# B&R Automation Studio project PLC code - cp (part 3)

#### Alarms.st
```iecst
ACTION Alarms:

	IF EDGEPOS(gDryer.AlSummary.xAlarmCritical) THEN
		MpAlarmXSet(gAlrCore, 'Dryer.Alarm.GenCritical');
	ELSIF EDGENEG(gDryer.AlSummary.xAlarmCritical) THEN
		MpAlarmXReset(gAlrCore, 'Dryer.Alarm.GenCritical');
	END_IF

	IF EDGEPOS(gDryer.AlSummary.xAlarmStop) THEN
		MpAlarmXSet(gAlrCore, 'Dryer.Alarm.GenStop');
	ELSIF EDGENEG(gDryer.AlSummary.xAlarmStop) THEN
		MpAlarmXReset(gAlrCore, 'Dryer.Alarm.GenStop');
	END_IF

	IF EDGEPOS(gDryer.Al.xAlrStopDrying) THEN
		MpAlarmXSet(gAlrCore, 'Dryer.Alarm.GenStopDrying');
	ELSIF EDGENEG(gDryer.Al.xAlrStopDrying) THEN
		MpAlarmXReset(gAlrCore, 'Dryer.Alarm.GenStopDrying');
	END_IF

	IF EDGEPOS(gDryer.Al.Alarm.xFanBreakers) THEN
		MpAlarmXSet(gAlrCore, 'Dryer.Alarm.FanBreakers');
	ELSIF EDGENEG(gDryer.Al.Alarm.xFanBreakers) THEN
		MpAlarmXReset(gAlrCore, 'Dryer.Alarm.FanBreakers');
	END_IF

	IF EDGEPOS(gDryer.Al.Alarm.xFan24Vdc) THEN
		MpAlarmXSet(gAlrCore, 'Dryer.Alarm.FansPsu');
	ELSIF EDGENEG(gDryer.Al.Alarm.xFan24Vdc) THEN
		MpAlarmXReset(gAlrCore, 'Dryer.Alarm.FansPsu');
	END_IF

	IF EDGEPOS(gDryer.Al.Alarm.xMain24Vdc) THEN
		MpAlarmXSet(gAlrCore, 'Dryer.Alarm.MainPsu');
	ELSIF EDGENEG(gDryer.Al.Alarm.xMain24Vdc) THEN
		MpAlarmXReset(gAlrCore, 'Dryer.Alarm.MainPsu');
	END_IF

	IF EDGEPOS(gDryer.Al.Alarm.xAlarmMountedMedia) THEN
		MpAlarmXSet(gAlrCore, 'Dryer.Alarm.MountedMedia');
	ELSIF EDGENEG(gDryer.Al.Alarm.xAlarmMountedMedia) THEN
		MpAlarmXReset(gAlrCore, 'Dryer.Alarm.MountedMedia');
	END_IF

	IF EDGEPOS(gDryer.Al.Alarm.Safety.xEStopFront) THEN
		MpAlarmXSet(gAlrCore, 'Dryer.Alarm.EstopFront');
	ELSIF EDGENEG(gDryer.Al.Alarm.Safety.xEStopFront) THEN
		MpAlarmXReset(gAlrCore, 'Dryer.Alarm.EstopFront');
	END_IF

	IF EDGEPOS(gDryer.Al.Alarm.Safety.xEStopRear) THEN
		MpAlarmXSet(gAlrCore, 'Dryer.Alarm.EstopRear');
	ELSIF EDGENEG(gDryer.Al.Alarm.Safety.xEStopRear) THEN
		MpAlarmXReset(gAlrCore, 'Dryer.Alarm.EstopRear');
	END_IF

	IF EDGEPOS(gDryer.Al.Alarm.Safety.xRemoteEStop) THEN
		MpAlarmXSet(gAlrCore, 'Dryer.Alarm.EstopRemote');
	ELSIF EDGENEG(gDryer.Al.Alarm.Safety.xRemoteEStop) THEN
		MpAlarmXReset(gAlrCore, 'Dryer.Alarm.EstopRemote');
	END_IF

	IF EDGEPOS(gDryer.Al.Alarm.xAlrWrongPhysConf) THEN
		MpAlarmXSet(gAlrCore, 'Dryer.Alarm.WrongPhysConfig');
	ELSIF EDGENEG(gDryer.Al.Alarm.xAlrWrongPhysConf) THEN
		MpAlarmXReset(gAlrCore, 'Dryer.Alarm.WrongPhysConfig');
	END_IF

	IF EDGEPOS(gDryer.Al.Alarm.xAlrBeltOvertorque) THEN
		MpAlarmXSet(gAlrCore, 'Dryer.Alarm.OvertorqueBelt');
	ELSIF EDGENEG(gDryer.Al.Alarm.xAlrBeltOvertorque) THEN
		MpAlarmXReset(gAlrCore, 'Dryer.Alarm.OvertorqueBelt');
	END_IF

	IF EDGEPOS(gDryer.Al.Alarm.xAlrBeltOverTempFast) THEN
		MpAlarmXSet(gAlrCore, 'Dryer.Alarm.OverTempBeltFast');
	ELSIF EDGENEG(gDryer.Al.Alarm.xAlrBeltOverTempFast) THEN
		MpAlarmXReset(gAlrCore, 'Dryer.Alarm.OverTempBeltFast');
	END_IF

	IF EDGEPOS(gDryer.Al.Alarm.xAlrBeltOverTempSlow) THEN
		MpAlarmXSet(gAlrCore, 'Dryer.Alarm.OverTempBeltSlow');
	ELSIF EDGENEG(gDryer.Al.Alarm.xAlrBeltOverTempSlow) THEN
		MpAlarmXReset(gAlrCore, 'Dryer.Alarm.OverTempBeltSlow');
	END_IF

	IF EDGEPOS(gDryer.Al.Warning.xFanBreakersHighLoad) THEN
		MpAlarmXSet(gAlrCore, 'Dryer.Alarm.FansPsu80');
	ELSIF EDGENEG(gDryer.Al.Warning.xFanBreakersHighLoad) THEN
		MpAlarmXReset(gAlrCore, 'Dryer.Alarm.FansPsu80');
	END_IF

	IF EDGEPOS(gDryer.Al.Warning.xMountedMediaInside) THEN
		MpAlarmXSet(gAlrCore, 'Dryer.Warning.MountedMediaInside');
	ELSIF EDGENEG(gDryer.Al.Warning.xMountedMediaInside) THEN
		MpAlarmXReset(gAlrCore, 'Dryer.Warning.MountedMediaInside');
	END_IF

	IF EDGEPOS(gDryer.Al.Warning.xBeltSensorError) THEN
		MpAlarmXSet(gAlrCore, 'Dryer.Warning.BeltTempSensError');
	ELSIF EDGENEG(gDryer.Al.Warning.xBeltSensorError) THEN
		MpAlarmXReset(gAlrCore, 'Dryer.Warning.BeltTempSensError');
	END_IF

	IF EDGEPOS(gDryer.Al.Warning.xBoardInSensorError) THEN
		MpAlarmXSet(gAlrCore, 'Dryer.Warning.BoardInTempSensError');
	ELSIF EDGENEG(gDryer.Al.Warning.xBoardInSensorError) THEN
		MpAlarmXReset(gAlrCore, 'Dryer.Warning.BoardInTempSensError');
	END_IF

	IF EDGEPOS(gDryer.Al.Warning.xBoardOutSensorError) THEN
		MpAlarmXSet(gAlrCore, 'Dryer.Warning.BoardOutTempSensError');
	ELSIF EDGENEG(gDryer.Al.Warning.xBoardOutSensorError) THEN
		MpAlarmXReset(gAlrCore, 'Dryer.Warning.BoardOutTempSensError');
	END_IF

	IF EDGEPOS(gDryer.Al.Warning.xAirBlowerInputSensorError) THEN
		MpAlarmXSet(gAlrCore, 'Dryer.Warning.AirBlowerInTempSensError');
	ELSIF EDGENEG(gDryer.Al.Warning.xAirBlowerInputSensorError) THEN
		MpAlarmXReset(gAlrCore, 'Dryer.Warning.AirBlowerInTempSensError');
	END_IF

	IF EDGEPOS(gDryer.Al.Warning.xAirBlowerOutputSensorError) THEN
		MpAlarmXSet(gAlrCore, 'Dryer.Warning.AirBlowerOutTempSensError');
	ELSIF EDGENEG(gDryer.Al.Warning.xAirBlowerOutputSensorError) THEN
		MpAlarmXReset(gAlrCore, 'Dryer.Warning.AirBlowerOutTempSensError');
	END_IF

	IF EDGEPOS(gDryer.Al.Warning.xFrontDoorOpened) THEN
		MpAlarmXSet(gAlrCore, 'Dryer.Warning.FrontDoorOpened');
	ELSIF EDGENEG(gDryer.Al.Warning.xFrontDoorOpened) THEN
		MpAlarmXReset(gAlrCore, 'Dryer.Warning.FrontDoorOpened');
	END_IF

	IF EDGEPOS(gDryer.Al.Warning.xRearDoorOpened) THEN
		MpAlarmXSet(gAlrCore, 'Dryer.Warning.RearDoorOpened');
	ELSIF EDGENEG(gDryer.Al.Warning.xRearDoorOpened) THEN
		MpAlarmXReset(gAlrCore, 'Dryer.Warning.RearDoorOpened');
	END_IF

	IF EDGEPOS(gDryer.Al.Warning.xBentMedia) THEN
		MpAlarmXSet(gAlrCore, 'Dryer.Warning.BentMedia');
	ELSIF EDGENEG(gDryer.Al.Warning.xBentMedia) THEN
		MpAlarmXReset(gAlrCore, 'Dryer.Warning.BentMedia');
	END_IF

	IF EDGEPOS(gDryer.Al.Warning.xNotEnabledMovement) THEN
		MpAlarmXSet(gAlrCore, 'Dryer.Warning.NotMovementEnabled');
	ELSIF EDGENEG(gDryer.Al.Warning.xNotEnabledMovement) THEN
		MpAlarmXReset(gAlrCore, 'Dryer.Warning.NotMovementEnabled');
	END_IF

	IF EDGEPOS(gDryer.Al.Warning.xKeyMantenanceActive) THEN
		MpAlarmXSet(gAlrCore, 'Dryer.Warning.KeyMantenance');
	ELSIF EDGENEG(gDryer.Al.Warning.xKeyMantenanceActive) THEN
		MpAlarmXReset(gAlrCore, 'Dryer.Warning.KeyMantenance');
	END_IF

	IF EDGEPOS(gDryer.Al.Warning.xJamLowCrash) THEN
		MpAlarmXSet(gAlrCore, 'Dryer.Warning.JamLowCrash');
	ELSIF EDGENEG(gDryer.Al.Warning.xJamLowCrash) THEN
		MpAlarmXReset(gAlrCore, 'Dryer.Warning.JamLowCrash');
	END_IF

	IF EDGEPOS(gBelt.Al.xAnyDriveAlarm) THEN
		MpAlarmXSet(gAlrCore, 'Dryer.Alarm.BeltAnyDriveAlarm');
	ELSIF EDGENEG(gBelt.Al.xAnyDriveAlarm) THEN
		MpAlarmXReset(gAlrCore, 'Dryer.Alarm.BeltAnyDriveAlarm');
	END_IF

	IF EDGEPOS(gBelt.Al.xAlrPowerBeltError) THEN
		MpAlarmXSet(gAlrCore, 'Dryer.Alarm.BeltAlrPowerBeltError');
	ELSIF EDGENEG(gBelt.Al.xAlrPowerBeltError) THEN
		MpAlarmXReset(gAlrCore, 'Dryer.Alarm.BeltAlrPowerBeltError');
	END_IF

	IF EDGEPOS(gBelt.Al.xAlrComDrive) THEN
		MpAlarmXSet(gAlrCore, 'Dryer.Alarm.BeltAlrComDrive');
	ELSIF EDGENEG(gBelt.Al.xAlrComDrive) THEN
		MpAlarmXReset(gAlrCore, 'Dryer.Alarm.BeltAlrComDrive');
	END_IF

	IF EDGEPOS(gBelt.Al.xAlrProtDrive) THEN
		MpAlarmXSet(gAlrCore, 'Dryer.Alarm.BeltAlrProtDrive');
	ELSIF EDGENEG(gBelt.Al.xAlrProtDrive) THEN
		MpAlarmXReset(gAlrCore, 'Dryer.Alarm.BeltAlrProtDrive');
	END_IF

	IF EDGEPOS(gBelt.Al.xAlrOverTorque) THEN
		MpAlarmXSet(gAlrCore, 'Dryer.Alarm.BeltAlrOverTorque');
	ELSIF EDGENEG(gBelt.Al.xAlrOverTorque) THEN
		MpAlarmXReset(gAlrCore, 'Dryer.Alarm.BeltAlrOverTorque');
	END_IF

	IF EDGEPOS(gBelt.Al.xBeltMotorTemp) THEN
		MpAlarmXSet(gAlrCore, 'Dryer.Alarm.BeltBeltMotorTemp');
	ELSIF EDGENEG(gBelt.Al.xBeltMotorTemp) THEN
		MpAlarmXReset(gAlrCore, 'Dryer.Alarm.BeltBeltMotorTemp');
	END_IF

	IF EDGEPOS(gBelt.Al.xBeltDriverTemp) THEN
		MpAlarmXSet(gAlrCore, 'Dryer.Alarm.BeltBeltDriverTemp');
	ELSIF EDGENEG(gBelt.Al.xBeltDriverTemp) THEN
		MpAlarmXReset(gAlrCore, 'Dryer.Alarm.BeltBeltDriverTemp');
	END_IF

	IF EDGEPOS(gBelt.Al.xAxisLengthNotDefined) THEN
		MpAlarmXSet(gAlrCore, 'Dryer.Alarm.BeltNoPerimeter');
	ELSIF EDGENEG(gBelt.Al.xAxisLengthNotDefined) THEN
		MpAlarmXReset(gAlrCore, 'Dryer.Alarm.BeltNoPerimeter');
	END_IF

	IF EDGEPOS(gBelt.Al.xGearBoxNotDefined) THEN
		MpAlarmXSet(gAlrCore, 'Dryer.Alarm.BeltNoGearBox');
	ELSIF EDGENEG(gBelt.Al.xGearBoxNotDefined) THEN
		MpAlarmXReset(gAlrCore, 'Dryer.Alarm.BeltNoGearBox');
	END_IF

	IF EDGEPOS(gBelt.Al.xWrnOverTorq) THEN
		MpAlarmXSet(gAlrCore, 'Dryer.Alarm.xWarningOvertoque');
	ELSIF EDGENEG(gBelt.Al.xWrnOverTorq) THEN
		MpAlarmXReset(gAlrCore, 'Dryer.Alarm.xWarningOvertoque');
	END_IF

	IF EDGEPOS(gSimpleBlock[1].Al.xAlrBarMtrNoRef) THEN
		MpAlarmXSet(gAlrCore, 'Dryer.Alarm.SblockNotReferenced');
	ELSIF EDGENEG(gSimpleBlock[1].Al.xAlrBarMtrNoRef) THEN
		MpAlarmXReset(gAlrCore, 'Dryer.Alarm.SblockNotReferenced');
	END_IF

	IF EDGEPOS(gSimpleBlock[1].Al.xAlrComBarMtr) THEN
		MpAlarmXSet(gAlrCore, 'Dryer.Alarm.SblockNotCommsDrive');
	ELSIF EDGENEG(gSimpleBlock[1].Al.xAlrComBarMtr) THEN
		MpAlarmXReset(gAlrCore, 'Dryer.Alarm.SblockNotCommsDrive');
	END_IF

	IF EDGEPOS(gSimpleBlock[1].Al.xAlrDriveProtection) THEN
		MpAlarmXSet(gAlrCore, 'Dryer.Alarm.SblockDriveBreaker');
	ELSIF EDGENEG(gSimpleBlock[1].Al.xAlrDriveProtection) THEN
		MpAlarmXReset(gAlrCore, 'Dryer.Alarm.SblockDriveBreaker');
	END_IF

	IF EDGEPOS(gSimpleBlock[1].Al.xAlrReferenceIncoherence) THEN
		MpAlarmXSet(gAlrCore, 'Dryer.Alarm.SblockHomeSensorError');
	ELSIF EDGENEG(gSimpleBlock[1].Al.xAlrReferenceIncoherence) THEN
		MpAlarmXReset(gAlrCore, 'Dryer.Alarm.SblockHomeSensorError');
	END_IF

	IF EDGEPOS(gSimpleBlock[1].Al.xAlrCheckHomingSensor) THEN
		MpAlarmXSet(gAlrCore, 'Dryer.Alarm.SblockCheckHomeSensor');
	ELSIF EDGENEG(gSimpleBlock[1].Al.xAlrCheckHomingSensor) THEN
		MpAlarmXReset(gAlrCore, 'Dryer.Alarm.SblockCheckHomeSensor');
	END_IF

	IF EDGEPOS(gSimpleBlock[1].Al.xBarMotorTemp) THEN
		MpAlarmXSet(gAlrCore, 'Dryer.Alarm.SblockMotorTemp');
	ELSIF EDGENEG(gSimpleBlock[1].Al.xBarMotorTemp) THEN
		MpAlarmXReset(gAlrCore, 'Dryer.Alarm.SblockMotorTemp');
	END_IF

	IF EDGEPOS(gSimpleBlock[1].Al.xBarDriverTemp) THEN
		MpAlarmXSet(gAlrCore, 'Dryer.Alarm.SblockDriveTemp');
	ELSIF EDGENEG(gSimpleBlock[1].Al.xBarDriverTemp) THEN
		MpAlarmXReset(gAlrCore, 'Dryer.Alarm.SblockDriveTemp');
	END_IF

	IF EDGEPOS(gTransVacuum[1].Alarms.xAlrVacuumSensor) THEN
		MpAlarmXSet(gAlrCore, 'Dryer.Alarm.VaccSensor');
	ELSIF EDGENEG(gTransVacuum[1].Alarms.xAlrVacuumSensor) THEN
		MpAlarmXReset(gAlrCore, 'Dryer.Alarm.VaccSensor');
	END_IF

	IF EDGEPOS(gTransVacuum[1].Alarms.xAlrCommsBlower[1]) THEN
		MpAlarmXSet(gAlrCore, 'Dryer.Alarm.VaccBlowerComsInput');
	ELSIF EDGENEG(gTransVacuum[1].Alarms.xAlrCommsBlower[1]) THEN
		MpAlarmXReset(gAlrCore, 'Dryer.Alarm.VaccBlowerComsInput');
	END_IF

	IF EDGEPOS(gTransVacuum[1].Alarms.xAlrCommsBlower[2]) THEN
		MpAlarmXSet(gAlrCore, 'Dryer.Alarm.VaccBlowerComsOutput');
	ELSIF EDGENEG(gTransVacuum[1].Alarms.xAlrCommsBlower[2]) THEN
		MpAlarmXReset(gAlrCore, 'Dryer.Alarm.VaccBlowerComsOutput');
	END_IF

	IF EDGEPOS(gTransVacuum[1].Alarms.xAlrBlowerCB[1]) THEN
		MpAlarmXSet(gAlrCore, 'Dryer.Alarm.VaccBlowerProtInput');
	ELSIF EDGENEG(gTransVacuum[1].Alarms.xAlrBlowerCB[1]) THEN
		MpAlarmXReset(gAlrCore, 'Dryer.Alarm.VaccBlowerProtInput');
	END_IF

	IF EDGEPOS(gTransVacuum[1].Alarms.xAlrBlowerCB[2]) THEN
		MpAlarmXSet(gAlrCore, 'Dryer.Alarm.VaccBlowerProtOutput');
	ELSIF EDGENEG(gTransVacuum[1].Alarms.xAlrBlowerCB[2]) THEN
		MpAlarmXReset(gAlrCore, 'Dryer.Alarm.VaccBlowerProtOutput');
	END_IF

	IF EDGEPOS(gTransVacuum[1].Alarms.xAlrBlowerError[1]) THEN
		MpAlarmXSet(gAlrCore, 'Dryer.Alarm.VaccBlowerErrorInput');
	ELSIF EDGENEG(gTransVacuum[1].Alarms.xAlrBlowerError[1]) THEN
		MpAlarmXReset(gAlrCore, 'Dryer.Alarm.VaccBlowerErrorInput');
	END_IF

	IF EDGEPOS(gTransVacuum[1].Alarms.xAlrBlowerError[2]) THEN
		MpAlarmXSet(gAlrCore, 'Dryer.Alarm.VaccBlowerErrorOutput');
	ELSIF EDGENEG(gTransVacuum[1].Alarms.xAlrBlowerError[2]) THEN
		MpAlarmXReset(gAlrCore, 'Dryer.Alarm.VaccBlowerErrorOutput');
	END_IF

	IF EDGEPOS(gTransVacuum[1].Alarms.xAlrBlowerNotRunning[1]) THEN
		MpAlarmXSet(gAlrCore, 'Dryer.Alarm.VaccBlowerNotRunningInput');
	ELSIF EDGENEG(gTransVacuum[1].Alarms.xAlrBlowerNotRunning[1]) THEN
		MpAlarmXReset(gAlrCore, 'Dryer.Alarm.VaccBlowerNotRunningInput');
	END_IF

	IF EDGEPOS(gTransVacuum[1].Alarms.xAlrBlowerNotRunning[2]) THEN
		MpAlarmXSet(gAlrCore, 'Dryer.Alarm.VaccBlowerNotRunningOutput');
	ELSIF EDGENEG(gTransVacuum[1].Alarms.xAlrBlowerNotRunning[2]) THEN
		MpAlarmXReset(gAlrCore, 'Dryer.Alarm.VaccBlowerNotRunningOutput');
	END_IF

	IF EDGEPOS(gNirAdphos.Alarms.xSafetyError) THEN
		MpAlarmXSet(gAlrCore, 'Dryer.Alarm.NIRSafetyError');
	ELSIF EDGENEG(gNirAdphos.Alarms.xSafetyError) THEN
		MpAlarmXReset(gAlrCore, 'Dryer.Alarm.NIRSafetyError');
	END_IF

	IF EDGEPOS(gNirAdphos.Alarms.xFault) THEN
		MpAlarmXSet(gAlrCore, 'Dryer.Alarm.NIRFault');
	ELSIF EDGENEG(gNirAdphos.Alarms.xFault) THEN
		MpAlarmXReset(gAlrCore, 'Dryer.Alarm.NIRFault');
	END_IF

	IF EDGEPOS(gNirAdphos.Alarms.xCommsError) THEN
		MpAlarmXSet(gAlrCore, 'Dryer.Alarm.NIRComsError');
	ELSIF EDGENEG(gNirAdphos.Alarms.xCommsError) THEN
		MpAlarmXReset(gAlrCore, 'Dryer.Alarm.NIRComsError');
	END_IF

	IF EDGEPOS(gNirAdphos.Alarms.xInletHumiditySensorError) THEN
		MpAlarmXSet(gAlrCore, 'Dryer.Alarm.NIRInletHumiditySensError');
	ELSIF EDGENEG(gNirAdphos.Alarms.xInletHumiditySensorError) THEN
		MpAlarmXReset(gAlrCore, 'Dryer.Alarm.NIRInletHumiditySensError');
	END_IF

	IF EDGEPOS(gNirAdphos.Alarms.xInletTempSensorError) THEN
		MpAlarmXSet(gAlrCore, 'Dryer.Alarm.NIRInletTempSensError');
	ELSIF EDGENEG(gNirAdphos.Alarms.xInletTempSensorError) THEN
		MpAlarmXReset(gAlrCore, 'Dryer.Alarm.NIRInletTempSensError');
	END_IF

	IF EDGEPOS(gJamDetect[1].Alarms.xAlrJamCrash[1]) THEN
		MpAlarmXSet(gAlrCore, 'Dryer.Alarm.JamInputNIR1');
	ELSIF EDGENEG(gJamDetect[1].Alarms.xAlrJamCrash[1]) THEN
		MpAlarmXReset(gAlrCore, 'Dryer.Alarm.JamInputNIR1');
	END_IF

	IF EDGEPOS(gJamDetect[1].Alarms.xAlrJamCrash[2]) THEN
		MpAlarmXSet(gAlrCore, 'Dryer.Alarm.JamOutputNIR1');
	ELSIF EDGENEG(gJamDetect[1].Alarms.xAlrJamCrash[2]) THEN
		MpAlarmXReset(gAlrCore, 'Dryer.Alarm.JamOutputNIR1');
	END_IF

	IF EDGEPOS(gJamDetect[1].Alarms.xAlrJamCrash[3]) THEN
		MpAlarmXSet(gAlrCore, 'Dryer.Alarm.JamInputNIR2');
	ELSIF EDGENEG(gJamDetect[1].Alarms.xAlrJamCrash[3]) THEN
		MpAlarmXReset(gAlrCore, 'Dryer.Alarm.JamInputNIR2');
	END_IF

	IF EDGEPOS(gJamDetect[1].Alarms.xAlrJamCrash[4]) THEN
		MpAlarmXSet(gAlrCore, 'Dryer.Alarm.JamOutputNIR2');
	ELSIF EDGENEG(gJamDetect[1].Alarms.xAlrJamCrash[4]) THEN
		MpAlarmXReset(gAlrCore, 'Dryer.Alarm.JamOutputNIR2');
	END_IF

	IF EDGEPOS(gNirAdphos.Alarms.Jam[1].xRear) THEN
		MpAlarmXSet(gAlrCore, 'Dryer.Alarm.JamRearNIR1');
	ELSIF EDGENEG(gNirAdphos.Alarms.Jam[1].xRear) THEN
		MpAlarmXReset(gAlrCore, 'Dryer.Alarm.JamRearNIR1');
	END_IF

	IF EDGEPOS(gNirAdphos.Alarms.Jam[2].xRear) THEN
		MpAlarmXSet(gAlrCore, 'Dryer.Alarm.JamRearNIR2');
	ELSIF EDGENEG(gNirAdphos.Alarms.Jam[2].xRear) THEN
		MpAlarmXReset(gAlrCore, 'Dryer.Alarm.JamRearNIR2');
	END_IF

	IF EDGEPOS(gNirAdphos.Alarms.Jam[1].xMechCross) THEN
		MpAlarmXSet(gAlrCore, 'Dryer.Alarm.JamMechCrossNIR1');
	ELSIF EDGENEG(gNirAdphos.Alarms.Jam[1].xMechCross) THEN
		MpAlarmXReset(gAlrCore, 'Dryer.Alarm.JamMechCrossNIR1');
	END_IF

	IF EDGEPOS(gNirAdphos.Alarms.Jam[2].xMechCross) THEN
		MpAlarmXSet(gAlrCore, 'Dryer.Alarm.JamMechCrossNIR2');
	ELSIF EDGENEG(gNirAdphos.Alarms.Jam[2].xMechCross) THEN
		MpAlarmXReset(gAlrCore, 'Dryer.Alarm.JamMechCrossNIR2');
	END_IF

	IF EDGEPOS(gNirAdphos.Alarms.xMaxSurfaceTempModule[1]) THEN
		MpAlarmXSet(gAlrCore, 'Dryer.Alarm.NIRSurfaceTemp1');
	ELSIF EDGENEG(gNirAdphos.Alarms.xMaxSurfaceTempModule[1]) THEN
		MpAlarmXReset(gAlrCore, 'Dryer.Alarm.NIRSurfaceTemp1');
	END_IF

	IF EDGEPOS(gNirAdphos.Alarms.xMaxSurfaceTempModule[2]) THEN
		MpAlarmXSet(gAlrCore, 'Dryer.Alarm.NIRSurfaceTemp2');
	ELSIF EDGENEG(gNirAdphos.Alarms.xMaxSurfaceTempModule[2]) THEN
		MpAlarmXReset(gAlrCore, 'Dryer.Alarm.NIRSurfaceTemp2');
	END_IF

	IF EDGEPOS(gNirAdphos.Alarms.xSurfaceTempModuleSensorError[1]) THEN
		MpAlarmXSet(gAlrCore, 'Dryer.Alarm.NIRSurfaceTempSensErr1');
	ELSIF EDGENEG(gNirAdphos.Alarms.xSurfaceTempModuleSensorError[1]) THEN
		MpAlarmXReset(gAlrCore, 'Dryer.Alarm.NIRSurfaceTempSensErr1');
	END_IF

	IF EDGEPOS(gNirAdphos.Alarms.xSurfaceTempModuleSensorError[2]) THEN
		MpAlarmXSet(gAlrCore, 'Dryer.Alarm.NIRSurfaceTempSensErr2');
	ELSIF EDGENEG(gNirAdphos.Alarms.xSurfaceTempModuleSensorError[2]) THEN
		MpAlarmXReset(gAlrCore, 'Dryer.Alarm.NIRSurfaceTempSensErr2');
	END_IF

	IF EDGEPOS(gNirAdphos.Alarms.BlockedFansModule[1].Fan[1]) THEN
		MpAlarmXSet(gAlrCore, 'Dryer.Alarm.BlockedFan1Nir1');
	ELSIF EDGENEG(gNirAdphos.Alarms.BlockedFansModule[1].Fan[1]) THEN
		MpAlarmXReset(gAlrCore, 'Dryer.Alarm.BlockedFan1Nir1');
	END_IF

	IF EDGEPOS(gNirAdphos.Alarms.BlockedFansModule[1].Fan[2]) THEN
		MpAlarmXSet(gAlrCore, 'Dryer.Alarm.BlockedFan2Nir1');
	ELSIF EDGENEG(gNirAdphos.Alarms.BlockedFansModule[1].Fan[2]) THEN
		MpAlarmXReset(gAlrCore, 'Dryer.Alarm.BlockedFan2Nir1');
	END_IF

	IF EDGEPOS(gNirAdphos.Alarms.BlockedFansModule[1].Fan[3]) THEN
		MpAlarmXSet(gAlrCore, 'Dryer.Alarm.BlockedFan3Nir1');
	ELSIF EDGENEG(gNirAdphos.Alarms.BlockedFansModule[1].Fan[3]) THEN
		MpAlarmXReset(gAlrCore, 'Dryer.Alarm.BlockedFan3Nir1');
	END_IF

	IF EDGEPOS(gNirAdphos.Alarms.BlockedFansModule[1].Fan[4]) THEN
		MpAlarmXSet(gAlrCore, 'Dryer.Alarm.BlockedFan4Nir1');
	ELSIF EDGENEG(gNirAdphos.Alarms.BlockedFansModule[1].Fan[4]) THEN
		MpAlarmXReset(gAlrCore, 'Dryer.Alarm.BlockedFan4Nir1');
	END_IF

	IF EDGEPOS(gNirAdphos.Alarms.BlockedFansModule[2].Fan[2]) THEN
		MpAlarmXSet(gAlrCore, 'Dryer.Alarm.BlockedFan1Nir2');
	ELSIF EDGENEG(gNirAdphos.Alarms.BlockedFansModule[2].Fan[2]) THEN
		MpAlarmXReset(gAlrCore, 'Dryer.Alarm.BlockedFan1Nir2');
	END_IF

	IF EDGEPOS(gNirAdphos.Alarms.BlockedFansModule[2].Fan[2]) THEN
		MpAlarmXSet(gAlrCore, 'Dryer.Alarm.BlockedFan2Nir2');
	ELSIF EDGENEG(gNirAdphos.Alarms.BlockedFansModule[2].Fan[2]) THEN
		MpAlarmXReset(gAlrCore, 'Dryer.Alarm.BlockedFan2Nir2');
	END_IF

	IF EDGEPOS(gNirAdphos.Alarms.BlockedFansModule[2].Fan[3]) THEN
		MpAlarmXSet(gAlrCore, 'Dryer.Alarm.BlockedFan3Nir2');
	ELSIF EDGENEG(gNirAdphos.Alarms.BlockedFansModule[2].Fan[3]) THEN
		MpAlarmXReset(gAlrCore, 'Dryer.Alarm.BlockedFan3Nir2');
	END_IF

	IF EDGEPOS(gNirAdphos.Alarms.BlockedFansModule[2].Fan[4]) THEN
		MpAlarmXSet(gAlrCore, 'Dryer.Alarm.BlockedFan4Nir2');
	ELSIF EDGENEG(gNirAdphos.Alarms.BlockedFansModule[2].Fan[4]) THEN
		MpAlarmXReset(gAlrCore, 'Dryer.Alarm.BlockedFan4Nir2');
	END_IF

	IF EDGEPOS(gArcLampGew.Alarms.xCommsError) THEN
		MpAlarmXSet(gAlrCore, 'Dryer.Alarm.ArcLampComsError');
	ELSIF EDGENEG(gArcLampGew.Alarms.xCommsError) THEN
		MpAlarmXReset(gAlrCore, 'Dryer.Alarm.ArcLampComsError');
	END_IF

	IF EDGEPOS(gArcLampGew.Alarms.Comms.xCredentialsError) THEN
		MpAlarmXSet(gAlrCore, 'Dryer.Alarm.ArcLampCredentialsError');
	ELSIF EDGENEG(gArcLampGew.Alarms.Comms.xCredentialsError) THEN
		MpAlarmXReset(gAlrCore, 'Dryer.Alarm.ArcLampCredentialsError');
	END_IF

	IF EDGEPOS(gArcLampGew.Alarms.Comms.xServerError) THEN
		MpAlarmXSet(gAlrCore, 'Dryer.Alarm.ArcLampInternalError');
	ELSIF EDGENEG(gArcLampGew.Alarms.Comms.xServerError) THEN
		MpAlarmXReset(gAlrCore, 'Dryer.Alarm.ArcLampInternalError');
	END_IF

	IF EDGEPOS(gArcLampGew.Alarms.xJam) THEN
		MpAlarmXSet(gAlrCore, 'Dryer.Alarm.ArcLampJam');
	ELSIF EDGENEG(gArcLampGew.Alarms.xJam) THEN
		MpAlarmXReset(gAlrCore, 'Dryer.Alarm.ArcLampJam');
	END_IF

	IF EDGEPOS(gArcLampGew.Status.Lamps[1].InAlarm) THEN
		MpAlarmXSet(gAlrCore, 'Dryer.Alarm.ArcLampAlarmLamp1');
	ELSIF EDGENEG(gArcLampGew.Status.Lamps[1].InAlarm) THEN
		MpAlarmXReset(gAlrCore, 'Dryer.Alarm.ArcLampAlarmLamp1');
	END_IF

	IF EDGEPOS(gArcLampGew.Status.Lamps[2].InAlarm) THEN
		MpAlarmXSet(gAlrCore, 'Dryer.Alarm.ArcLampAlarmLamp2');
	ELSIF EDGENEG(gArcLampGew.Status.Lamps[2].InAlarm) THEN
		MpAlarmXReset(gAlrCore, 'Dryer.Alarm.ArcLampAlarmLamp2');
	END_IF

	IF EDGEPOS(gThicknessCtrl.Alarms.CheckMedia[1]) THEN
		MpAlarmXSet(gAlrCore, 'Dryer.Alarm.CheckMediaExit1');
	ELSIF EDGENEG(gThicknessCtrl.Alarms.CheckMedia[1]) THEN
		MpAlarmXReset(gAlrCore, 'Dryer.Alarm.CheckMediaExit1');
	END_IF

	IF EDGEPOS(gThicknessCtrl.Alarms.CheckMedia[2]) THEN
		MpAlarmXSet(gAlrCore, 'Dryer.Alarm.CheckMediaExit2');
	ELSIF EDGENEG(gThicknessCtrl.Alarms.CheckMedia[2]) THEN
		MpAlarmXReset(gAlrCore, 'Dryer.Alarm.CheckMediaExit2');
	END_IF

END_ACTION
```

- DryerTextsAndAlarms.csv (not shown)

### Program Logical/Dryer/PhysicalMapping/PhysicalMapInputs

#### MappingInputs.st
```iecst
PROGRAM _CYCLIC

	//If in automation runtime, do not assign physical mapping
	IF gDryer.St.HwData.Family = FAMILY_BRAUTOMATIONRUNTIME THEN
		RETURN;
	END_IF

	CASE gDryer.Pt.MachineModel OF
		DryerType_NOZ2_NIR,
		DryerType_NOZ2_NIR_ARCLAMP:
			InputsDryerNoz2;

	END_CASE

END_PROGRAM
```

### Program Logical/Dryer/PhysicalMapping/PhysicalMapOutputs

#### OutputsDryerNoz2.st
```iecst
ACTION OutputsDryerNoz2:

	// X20DOF322_205 DIGITAL OUTPUTS
	X20DOF322_205.DOutput[1] := gNirAdphos.Signals.Out.xPowerOn;
	X20DOF322_205.DOutput[2] := gNirAdphos.Signals.Out.xProcess;
	X20DOF322_205.DOutput[3] := gNirAdphos.Signals.Out.xSafetyStop;
	X20DOF322_205.DOutput[4] := NOT gDryer.Out.xKeepSafetyNIR; //gArcLampGew.Signals.Out.xImpression;
	X20DOF322_205.DOutput[5] := gJamDetect[1].Outputs.xJamTestSignal[1];
	X20DOF322_205.DOutput[6] := gJamDetect[1].Outputs.xJamTestSignal[2];
	X20DOF322_205.DOutput[7] := gJamDetect[1].Outputs.xJamTestSignal[3];
	X20DOF322_205.DOutput[8] := gJamDetect[1].Outputs.xJamTestSignal[4];

	// X20DOF322_206 DIGITAL OUTPUTS
	X20DOF322_206.DOutput[1] := gDryer.Out.xLockFrontDoor;
	X20DOF322_206.DOutput[2] := gDryer.Out.xLockRearDoor;
	X20DOF322_206.DOutput[3] := gDryer.Out.xResetFanBreaker;
	X20DOF322_206.DOutput[4] := gDryer.Out.xResetHub;
	X20DOF322_206.DOutput[5] := gDryer.Out.xResetSwitch;
	X20DOF322_206.DOutput[6] := gDryer.AlSummary.xAlarmCritical OR gDryer.AlSummary.xAlarmStop;
	X20DOF322_206.DOutput[7] := FALSE;
	X20DOF322_206.DOutput[8] := FALSE;
	X20DOF322_206.DOutput[9] := FALSE;
	X20DOF322_206.DOutput[10] := FALSE;
	X20DOF322_206.DOutput[11] := gDryer.Out.xBuzzer;
	X20DOF322_206.DOutput[12] := gDryer.Out.xYellowLight;
	X20DOF322_206.DOutput[13] := gDryer.Out.xBlueLight;
	X20DOF322_206.DOutput[14] := gDryer.Out.xRedLight;
	X20DOF322_206.DOutput[15] := gDryer.Out.xWhiteLight;
	X20DOF322_206.DOutput[16] := gDryer.Out.xResetBlueLight;

	// X20AO4622_208 ANALOG OUTPUTS
	X20AO4622_208.AOutput[1] := gNirAdphos.Signals.Out.iBeltSpeed;
	X20AO4622_208.AOutput[2] := gArcLampGew.Signals.Out.iBeltSpeed;

END_ACTION
```

### Program Logical/Dryer/Sim/SimDryer (IEC)

#### SimDryer.st - Init, cyclic, exit code
```iecst
PROGRAM _INIT

	gDryer.In.xMain24VdcOK:=TRUE;
	gDryer.In.xFan24VdcOK:=TRUE;
	gDryer.In.xFanBreakersOK:=TRUE;
	gDryer.In.xFanBreakersWarning:=TRUE;

	gNirAdphos.Signals.In.iInletHumidityRaw := 20000;
	gNirAdphos.Signals.In.iInletTempRaw := 25000;

	gDryer.In.Temp.iBeltRaw := 10500;
	gDryer.In.Temp.iBoardInRaw := 10000;
	gDryer.In.Temp.iBoardOutRaw := 11000;
	gDryer.In.Temp.iAirBlowerInputRaw := 12000;
	gDryer.In.Temp.iAirBlowerOutputRaw := 12500;

	gDryer.In.Safety.xClosedFrontInput := TRUE;
	gDryer.In.Safety.xClosedFrontOutput := TRUE;
	gDryer.In.Safety.xClosedRearInput := TRUE;
	gDryer.In.Safety.xClosedRearOutput := TRUE;
	gDryer.In.Safety.xEStopFrontOK := TRUE;
	gDryer.In.Safety.xEStopRearOK := TRUE;
	gDryer.In.Safety.xMovementsEnabled := TRUE;
	gDryer.In.Safety.xRemoteEStopOK := TRUE;

	gDryerRemoteData.Signals.Safety.xClosedFrontInput := TRUE;
	gDryerRemoteData.Signals.Safety.xClosedFrontOutput := TRUE;
	gDryerRemoteData.Signals.Safety.xClosedRearInput := TRUE;
	gDryerRemoteData.Signals.Safety.xClosedRearOutput := TRUE;
	gDryerRemoteData.Signals.Safety.xEStopFrontOK := TRUE;
	gDryerRemoteData.Signals.Safety.xEStopRearOK := TRUE;
	gDryerRemoteData.Signals.Safety.xMovementsEnabled := TRUE;
	gDryerRemoteData.Signals.Safety.xRemoteEStopOK := TRUE;

	gDryerRemoteData.Signals.xBreakerOKBlowerInput := TRUE;
	gDryerRemoteData.Signals.xBreakerOKBlowerOutput := TRUE;

	//We need to write over the permanent var because is loaded during machine init
	//gPermanentBelt.xDriveProtectionOK:=TRUE;
	gBelt.parameters.xDriveProtectionOK:=TRUE;

	gAxisInverter[1].ElecSignals.In.xBreakerOK := TRUE;
	gAxisInverter[2].ElecSignals.In.xBreakerOK := TRUE;

	URLHost := '127.0.0.1';

	webClient.option := httpOPTION_HTTP_11;
	webClient.pHost := ADR(URLHost);
	webClient.pUri := ADR(URIHost);
	webClient.hostPort := 83;
	webClient.method := httpMETHOD_GET;

	webClient.pResponseHeader := ADR(ResponseHeader);
	webClient.pResponseData := ADR(ResponseData);
	webClient.responseDataSize := SIZEOF(ResponseData);
	webClient.pRequestData := ADR(RequestData);
	webClient.requestDataLen := SIZEOF(RequestData);

	gSimMachine.Parameters.DryerType := SIM_DRYER_NOZ2_NIR;
	gSimMachine.Parameters.xAutoMediaPresent := TRUE;

	gDryer.Pt.SW.Media.rThickness := 3.2;
	gDryer.Pt.SW.Media.rWidth := 1400;
	gDryer.Pt.SW.Media.rLength := 2500;
	gDryer.Pt.SW.Media.rCrossOffset := -700;
	gDryer.Pt.SW.Media.rDocWidth := 1400;
	gDryer.Pt.SW.Media.rDocLength := 2500;
	gDryer.Pt.SW.Media.rDocCrossOffset := -700;

	gSimDryer.Parameters.rGap := 400; //To simulate entering media

	// ###################################
	// END OF INIT CODE

END_PROGRAM

PROGRAM _CYCLIC

	//Define the inputs of the Machine depending the machine to Simulate
	CASE gSimMachine.Parameters.DryerType OF
		SIM_DRYER_NOZ2_NIR_ARCLAMP:
			gDryer.In.iMachineModelCode:=3;
		SIM_DRYER_NOZ2_NIR:
			gDryer.In.iMachineModelCode:=2;
	END_CASE

	gDryer.In.Buttons.xManual := gDryer.In.xManual_GI;
	gDryer.In.Buttons.xZero := gDryer.In.xZero_GI;
	gDryer.In.Buttons.xAuto := gDryer.In.xAuto_GI;
	gDryer.In.Buttons.xStopBlowers := gDryer.In.Sw.xStopBlowers_GI;

	//Signal from the selector
	IF EDGEPOS(gDryer.In.Buttons.xManual) THEN
		gDryer.In.Buttons.xZero:=FALSE;
		gDryer.In.Buttons.xAuto:=FALSE;
	END_IF
	IF EDGEPOS(gDryer.In.Buttons.xZero) THEN
		gDryer.In.Buttons.xManual:=FALSE;
		gDryer.In.Buttons.xAuto:=FALSE;
	END_IF
	IF EDGEPOS(gDryer.In.Buttons.xAuto) THEN
		gDryer.In.Buttons.xManual:=FALSE;
		gDryer.In.Buttons.xZero:=FALSE;
	END_IF

	IF EDGE(gDryer.In.Sw.xReset_GI) THEN
		gDryer.In.Buttons.xReset:=gDryer.In.Sw.xReset_GI;
	END_IF

	IF EDGEPOS(gSimMachine.Commands.xToZero) THEN
		gDryer.In.Buttons.xZero:=TRUE;
		gDryer.In.Buttons.xManual:=FALSE;
		gDryer.In.Buttons.xAuto:=FALSE;

		simEventLog.Source := ELOG_TYPE_GENERAL;
		simEventLog.Severity:= ELOG_SEVERITY_INFO;
		simEventLog.Facility:= 0;
		simEventLog.ErrorCode:=0;
		simEventLog.Text := 'Machine going to Zero in Simulation';
		gEventLogLoader(EventData:=ADR(simEventLog));

	END_IF
	IF gSimMachine.Commands.xToZero AND gDryer.St.Mode.xZero THEN
		gSimMachine.Commands.xToZero:=FALSE;
	END_IF

	IF EDGEPOS(gSimMachine.Commands.xToManual) AND gDryer.St.Mode.xManual THEN
		gSimMachine.Commands.xToManual:=FALSE;
	END_IF
	IF EDGEPOS(gSimMachine.Commands.xToManual) THEN
		gDryer.In.Buttons.xZero:=FALSE;
		gDryer.In.Buttons.xManual:=TRUE;
		gDryer.In.Buttons.xAuto:=FALSE;
		gDryer.In.Buttons.xReset:=TRUE;
	END_IF
	IF gSimMachine.Commands.xToManual AND gDryer.St.Mode.xManual THEN
		gSimMachine.Commands.xToManual:=FALSE;
		gDryer.In.Buttons.xReset:=FALSE;
	END_IF

	IF EDGEPOS(gSimMachine.Commands.xToAuto) AND gDryer.St.Mode.xAuto THEN
		gSimMachine.Commands.xToAuto:=FALSE;
	END_IF
	IF EDGEPOS(gSimMachine.Commands.xToAuto) THEN
		gDryer.In.Buttons.xZero:=FALSE;
		gDryer.In.Buttons.xManual:=FALSE;
		gDryer.In.Buttons.xAuto:=TRUE;
		gDryer.In.Buttons.xReset:=TRUE;
	END_IF
	IF gSimMachine.Commands.xToAuto AND gDryer.St.Mode.xAuto THEN
		gSimMachine.Commands.xToAuto:=FALSE;
		gDryer.In.Buttons.xReset:=FALSE;
	END_IF

	IF EDGEPOS(gSimMachine.Commands.Media.xMediaPresent) THEN
		//TOBEIMPLEMENTED
	END_IF
	IF EDGENEG(gSimMachine.Commands.Media.xMediaPresent) THEN
		//TOBEIMPLEMENTED
	END_IF

	tonSimMediaAuto.IN := gSimMachine.Parameters.xAutoMediaPresent AND gDryer.St.Mode.xAuto AND (gDryer.St.DryerState = DRYERMACH_DRYING OR gDryer.St.DryerState = DRYERMACH_STARTING);
	IF gBelt.states.rCurrentSpeed > 1 THEN
		tonSimMediaAuto.PT := REAL_TO_TIME(60 * (gDryer.Pt.SW.Media.rLength + gSimDryer.Parameters.rGap) / gBelt.states.rCurrentSpeed);
	ELSE
		tonSimMediaAuto.PT := t#3s; // default and previous value
	END_IF
	tonSimMediaAuto();

	IF gDryer.St.Mode.xAuto THEN
		//Starting system
		IF EDGEPOS(gDryer.St.DryerState = DRYERMACH_DRYING) OR EDGEPOS(tonSimMediaAuto.Q) THEN
			xSimulateMedia := TRUE;
		ELSIF EDGENEG(gDryer.St.DryerState = DRYERMACH_DRYING) THEN
			xSimulateMedia := FALSE;
		END_IF
	ELSE
		xSimulateMedia := FALSE;
	END_IF

	tonSimMedia.IN := xSimulateMedia AND NOT tonSimMedia.Q;
	IF gBelt.states.rCurrentSpeed = 0 THEN
		tonSimMedia.PT := t#3s;
	ELSE
		tonSimMedia.PT := REAL_TO_TIME(60 * (gDryer.Pt.SW.Media.rLength + gSimDryer.Parameters.rGap) / gBelt.states.rCurrentSpeed);
	END_IF
	tonSimMedia();

	IF EDGEPOS(tonSimMedia.Q) THEN
		gDryerLocalSignals.Signals.xMediaPresent := NOT gDryerLocalSignals.Signals.xMediaPresent;
		gBasicDetectMedia.Inputs.xMediaPresentL1 := NOT gBasicDetectMedia.Inputs.xMediaPresentL1;
	END_IF
	IF EDGENEG(xSimulateMedia) THEN
		gDryerLocalSignals.Signals.xMediaPresent := FALSE;
		gBasicDetectMedia.Inputs.xMediaPresentL1 := FALSE;
	END_IF

	// Not the best way to simulate the behaviour, maybe in the future we will need something more accurate
	gThicknessCtrl.Inputs.CheckMedia[1].xCheckFail := gThicknessCtrl.status.MediaPosition.xMediaInside;
	gThicknessCtrl.Inputs.CheckMedia[2].xCheckFail := gThicknessCtrl.status.MediaPosition.xMediaInside;

	//Configuration of the calling to the TestExecution

	IF xTestPrepareDryer THEN
		URIHost := '/WsTest/PrepareDryer';
	ELSIF xTestBeltTests THEN
		URIHost := '/WsTest/BeltTests';
	ELSIF xTestConsents THEN
		URIHost := '/WsTest/ConsentTests';
	ELSIF xTestCleaning THEN
		URIHost := '/WsTest/CleaningTests';
	ELSIF xTestLine THEN
		URIHost := '/WsTest/LineTests';
	END_IF

	webClient.enable:=TRUE;
	webClient.send:= xTestPrepareDryer OR xTestBeltTests OR xTestConsents OR xTestCleaning OR xTestLine;
	webClient();

	testMonitor.Enable:=TRUE;
	testMonitor();
	gTestsExec.testPassedAsserts := testMonitor.Informational.PassedAssertCounter;
	gTestsExec.testFailedAsserts := testMonitor.Informational.FailedAssertCounter;
	gTestsExec.xSometestFailedAsserts := testFailedAsserts > 0;
	gTestsExec.xAnyTestActive := testMonitor.TestActive;
	gTestsExec.xSimMachine := gDryer.St.HwData.Family = FAMILY_BRAUTOMATIONRUNTIME;

	gSimNirAdphos.Parameters.CurrentSpeed := gBelt.states.rCurrentSpeed;

	IF simMachineTypeEnumCopy<>gSimMachine.Parameters.MachineType THEN
		simMachineType := DINT_TO_INT(gSimMachine.Parameters.MachineType);
	END_IF
	IF simMachineType<>simMachineTypeCopy THEN
		gSimMachine.Parameters.MachineType := simMachineType;
	END_IF

	simMachineTypeCopy := simMachineType;
	simMachineTypeEnumCopy := gSimMachine.Parameters.MachineType;

	gDryer.In.xManual_GI := gDryer.In.Buttons.xManual;
	gDryer.In.xZero_GI := gDryer.In.Buttons.xZero;
	gDryer.In.xAuto_GI := gDryer.In.Buttons.xAuto;
	gDryer.In.Sw.xStopBlowers_GI := gDryer.In.Buttons.xStopBlowers;

END_PROGRAM

PROGRAM _EXIT
	gBelt; //Just to allow to watch it ;-)
	gEventLogManager; //Just here to be able to watch this var
END_PROGRAM
```

### SimDryer.typ
```iecst
TYPE
	SimDryerParameters_typ : 	STRUCT
		rGap : REAL;
	END_STRUCT;
	SimDryer_typ : 	STRUCT
		Parameters : SimDryerParameters_typ;
	END_STRUCT;
END_TYPE
```

### Package Logical/ExtPack/EFILib - Efi libs package

### Package Logical/ExtPack/EFILib/EFILib_v1 - Efi libs package

### Library Logical/ExtPack/EFILib/EFILib_v1/FBs (IEC) - Functional blocks
Depends on: standard, AsIecCon

#### Constants.var - Exported constants
```iecst
VAR CONSTANT
	FAMILY_BRAUTOMATIONRUNTIME : USINT := 4;
	FAMILY_BRX2X : USINT := 10;
	MOTOR_POSITIVE_AXIS : USINT := 0;
	MOTOR_NEGATIVE_AXIS : USINT := 1;
END_VAR
(**)
(*#############################
HTTP STATUS CODES*)
VAR CONSTANT
	HTTPSTATUS_OK : UINT := 200;
	HTTPSTATUS_BADREQUEST : UINT := 400;
	HTTPSTATUS_UNAUTORIZED : UINT := 401;
	HTTPSTATUS_NOTFOUND : UINT := 404;
	HTTPSTATUS_INTERNALSERVERERROR : UINT := 500;
END_VAR
(*#############################
MEDIA TRACKING*)
VAR CONSTANT
	MEDIATRACKING_UNKNOWN : SINT := -1; (*-1: MEDIATRACKING_UNKNOWN*)
	MEDIATRACKING_INVALID : SINT := 0; (*0: MEDIATRACKING_INVALID*)
	MEDIATRACKING_VALID : SINT := 1; (*1: MEDIATRACKING_VALID*)
END_VAR
```

#### IclaConstants.var
```iecst
VAR CONSTANT
	ICLAST_ERROR : UINT := 9;
	ICLAST_FAULTREACTION_ACTIVE : UINT := 8;
	ICLAST_QUICKSTOP_ACTIVE : UINT := 7;
	ICLAST_ENABLE_OPERATION : UINT := 6;
	ICLAST_READY_TO_SWITCH_ON : UINT := 4;
	ICLAST_SWITCH_ON_DISABLED : UINT := 3;
	ICLAST_NOTREADY_TO_SWITCH_ON : UINT := 2;
END_VAR
```

#### InksPublicConst.var - Global Ink Constant Vars
```iecst
VAR CONSTANT
	lc_iInkMineral : INT := 1;
	lc_iInkSolubleSalts : INT := 2;
	lc_iInkWater : INT := 4;
	lc_iInkUV : INT := 8;
	lc_iPrintHeadTtec : INT := 1; (*Printhead Toshiba*)
	lc_iPrintHeadX1003 : INT := 3; (*Printhead XSAAR*)
	lc_iPrintHeadX1003gs40 : INT := 6; (*Printhead XSAAR*)
	lc_iPrintHeadX2001 : INT := 7; (*Printhead XSAAR Dual Color*)
	lc_iPrintHeadX2001gs40 : INT := 8; (*Printhead XSAAR*)
	lc_iPrintHeadTtecXL : INT := 5; (*Printhead Toshiba L*)
	lc_iPrintHeadDimatics : INT := 4; (*Printhead Dimatics Manufacture. It is pendig to be defined in P4*)
	lc_iPrintHeadSK1536 : INT := 2; (*Printhead Seiko*)
	lc_iPrintHeadSK1536L : INT := 10; (*Printhead SeikoL*)
	lc_iPrintHeadSK1536W : INT := 9; (*Printhead Seiko Water*)
	lc_iPrintHeadSK1536LW : INT := 12; (*Printhead SeikoL Water*)
	INKS_DRIP_TIME_MAX : TIME := T#30S; (*Max value of DripTime in seconds*)
	lc_iPrintHeadKatana : INT := 13; (*Printhead Kyocera Katana*)
	lc_iPrintHeadRicoh : INT := 15;
END_VAR
```

#### FbCleanDelayControl.st - Gap delay control
```iecst
FUNCTION_BLOCK FbCleanDelayControl
	IF  (Doble) THEN

		// Calculo para linea doble
		IF T_delay_L1 > T_delay_L2 THEN
			T_delay1:=T#0S;
			T_delay2:=T_delay_L1 - T_delay_L2;
		ELSE
			T_delay1:=T_delay_L2 - T_delay_L1;
			T_delay2:=T#0S;
		END_IF;

		IF ( t_Gap<=0) THEN

			// No gap. Only doble line delay
			TON_1 (IN:= Start, PT:= T_delay1 );
			TON_5 (IN:= Start, PT:= T_delay2 );

			TON_4 (IN:= TON_1.Q, PT:= T_delay_L1);
			TON_6 (IN:= TON_5.Q, PT:= T_delay_L2);

			IF TON_4.Q AND TON_6.Q THEN
				End:= TRUE;
			ELSE
				End:= FALSE;
			END_IF

			IF 	(( T_delay_L1>0) OR ( T_delay_L2>0)) AND TON_1.Q THEN
				Out_L1:= TRUE;
			ELSE
				Out_L1:= FALSE;
			END_IF

			IF 	(( T_delay_L1>0) OR ( T_delay_L2>0)) AND TON_5.Q THEN
				Out_L2:= TRUE;
			ELSE
				Out_L2:= FALSE;
			END_IF

		ELSIF (t_Gap>0) THEN

			// With doble line gap
			TON_12 (IN:= (Start), PT:= T_delay1 );
			TON_14 (IN:=( Start), PT:= T_delay2 );

			TON_13 (IN:= TON_12.Q, PT:= T_delay_L1);
			TON_15 (IN:= TON_14.Q, PT:= T_delay_L2);

			IF TON_13.Q AND TON_15.Q THEN
				End:= TRUE;
			ELSE
				End:= FALSE;
			END_IF

			TON_9 (IN:=TON_12.Q, PT:=t_Gap);
			TON_16 (IN:=TON_14.Q, PT:= t_Gap);

			IF TON_12.Q AND NOT TON_9.Q THEN
				Out_L1:= TRUE;
			ELSE
				Out_L1:= FALSE;
			END_IF

			IF TON_14.Q AND NOT TON_16.Q THEN
				Out_L2:= TRUE;
			ELSE
				Out_L2:= FALSE;
			END_IF

		END_IF

	//////////////////////////////////////////////////////////
	// No Gap. Only single line delay
	// Pre_Stop only activated if the value is > 0
	//Jira Reference: CRETALEGO-1011
	//////////////////////////////////////////////////////////

	ELSIF  (NOT Doble) THEN
		TON_0 (IN:= ( (t_Gap<=0) AND Start), PT:= T_delay_L1);
		End:=TON_0.Q;

		IF ( t_Gap<=0) AND Start AND ( T_delay_L1>0) THEN
			Out_L1:= TRUE;
		ELSE
			Out_L1:= FALSE;
		END_IF

		//	With gap in single line
		IF ( t_Gap>0) THEN
			TON_3 (IN:= ( (t_Gap>0) AND Start), PT:= T_delay_L1);
			End:=TON_3.Q;
		END_IF

		TON_2 (IN:= ( t_Gap>0) AND Start, PT:= t_Gap);

		IF ( t_Gap>0) AND  Start AND NOT TON_2.Q THEN
			Out_L1:= TRUE;
		ELSE
			Out_L1:= FALSE;
		END_IF

	END_IF
END_FUNCTION_BLOCK
```

#### MotorDistanceCalculation.st - Distance in Units motor
```iecst
// It gets distance in pulses
//FUNCTION_BLOCK MotorDistanceCalculation
//
//	uiMotorDistanceInPulses :=  (uiSpDistance*uiPulsesPerRev / uiWheelPerimeter);
//
//END_FUNCTION_BLOCK
```

#### ComandBoolT.st
```iecst
(* TODO: Add your comment here *)
FUNCTION_BLOCK ComandBoolT

	IF Com = 1 THEN
		In := TRUE;
	END_IF

	IF Com = 0 THEN
		In := FALSE;
	END_IF

	IF In THEN
		Contador := Contador + 1;
	END_IF

	IF Contador >= 2 THEN
		In := FALSE;
		Contador := 0;
	END_IF

	Com := -1;
END_FUNCTION_BLOCK
```

#### Blink.st
```iecst
(* TODO: Add your comment here *)
FUNCTION_BLOCK Blink

	T_ON.PT:= T_Blink;
	T_ON.IN:= NOT T_OFF.Q;
	T_ON();

	T_OFF.IN:= T_ON.Q;
	T_OFF.PT:= T_Blink;
	T_OFF();

	Out:= T_ON.Q;

	VAR1:= TRUE;

END_FUNCTION_BLOCK
```

#### InterfaceNetworkCommands.st
```iecst
//FUNCTION_BLOCK InterfaceNetworkCommands
//// Pending to do reset SMC code (cyclic program) as FB
//
//END_FUNCTION_BLOCK
```

#### BlinkOnOff.st
```iecst
(* TODO: Add your comment here *)
FUNCTION_BLOCK BlinkOnOff
	TON_1(IN := xEnable AND NOT TON_2.Q, PT := tTimeOn );
	TON_2(IN := TON_1.Q, PT := tTimeOff );
	xOutput:= xEnable AND NOT TON_1.Q AND NOT TON_2.Q;
END_FUNCTION_BLOCK
```

#### SimAnalogProcess.st
```iecst
(* TODO: Add your comment here *)
FUNCTION_BLOCK SimAnalogProcess

	//Start with the initial value
	IF NOT xStarted THEN
		rPresentValue:=rInitialValue;
		xStarted:=TRUE;
	END_IF

	IF EDGEPOS(xUseNewValue) THEN
		xUseNewValue:=FALSE;
		rPresentValue:=rNewPresentValue;
	END_IF

	CASE AnalogType OF
		ANALOGSIM_LINEAR_POS, ANALOGSIM_EXPONENTIAL_POS:
			rSignalPerct := ABS(rMaxValue-rPresentValue)/ABS(rMaxValue-rMinValue);
		ANALOGSIM_LINEAR_NEG, ANALOGSIM_EXPONENTIAL_NEG:
			rSignalPerct := ABS(rPresentValue-rMinValue)/ABS(rMaxValue-rMinValue);
	END_CASE;

	//Calculate the next value
	CASE AnalogType OF

		ANALOGSIM_LINEAR_NEG, ANALOGSIM_LINEAR_POS:
			rPresentValue := rPresentValue - rA + rB * rActionControl;

		ANALOGSIM_EXPONENTIAL_POS:
			rPresentValue := rPresentValue + ABS(rA) * EXPT(rSignalPerct,2) - ABS(rB) * rActionControl;

		ANALOGSIM_EXPONENTIAL_NEG:
			rPresentValue := rPresentValue - ABS(rA) * EXPT(rSignalPerct,2) + ABS(rB) * rActionControl;

	END_CASE;

	//Limit the PV
	rPresentValue := LIMIT( rMinValue, rPresentValue, rMaxValue);

END_FUNCTION_BLOCK
```

### Library Logical/ExtPack/EFILib/EFILib_v1/Functions (IEC) - Functions

#### Functions.typ
```iecst
TYPE
	stPIDParam : 	STRUCT
		rKp : REAL;
		rTi : REAL;
		rKd : REAL;
		rTd : REAL;
		zFree : ARRAY[0..4]OF USINT;
	END_STRUCT;
	StPLC_Internal : 	STRUCT
		Blink_1s : Blink;
		Blink_2s : Blink;
		Blink_5s : Blink;
		Blink_10s : Blink;
		Blink_100ms : Blink;
		Blink_200ms : Blink;
		Blink_500ms : Blink;
		RestartInfo : RTInfo;
	END_STRUCT;
	StPLC : 	STRUCT
		xBlk_100ms : BOOL;
		xBlk_200ms : BOOL;
		xBlk_500ms : BOOL;
		xBlk_1s : BOOL;
		xBlk_2s : BOOL;
		xBlk_5s : BOOL;
		xBlk_10s : BOOL;
		xColdRestart : BOOL;
		xWarmRestart : BOOL;
		xDownloadRestart : BOOL;
		xFirst_Scan : BOOL;
		iZero : USINT;
		diCycleTime : UDINT := 0; (*Cycle time in microseconds*)
		iVarsVersion0 : UINT;
		iVarsVersion1 : UINT;
		iVarsVersion2 : UINT;
		iVarsVersion3 : UINT;
		iVersion0 : UINT;
		iVersion1 : UINT;
		iVersion2 : UINT;
		iVersion3 : UINT;
		sVersion : STRING[20];
		sLastPlcProgrammer : STRING[20];
		Internal : StPLC_Internal;
	END_STRUCT;
END_TYPE
```

#### Functions.fun - Exported functions and function blocks
```iecst
FUNCTION ComandBool : BOOL (*To be used with vars that remotely set or reset with an order of 1 or 0*) (*$GROUP=User,$CAT=User,$GROUPICON=User.png,$CATICON=User.png*)
	VAR_IN_OUT
		In : BOOL; (*The BOOL var set/reset by the command*)
		Com : INT; (*Command. 1 to set and 0 to reset. After a command, the function sets it to -1*)
	END_VAR
END_FUNCTION

FUNCTION ComandBoolEdge0 : BOOL (*To be used with vars that with an order of 1 are set to TRUE during one comms cycle*) (*$GROUP=User,$CAT=User,$GROUPICON=User.png,$CATICON=User.png*)
	VAR_IN_OUT
		In : BOOL; (*The BOOL var set/reset by the command*)
		Com : INT; (*Command. 1 to set and 0 to reset. After a command, the function sets it to -1*)
	END_VAR
END_FUNCTION

FUNCTION ComandBoolReset : BOOL (*To be used with vars that remotely RESET with an order of 1*) (*$GROUP=User,$CAT=User,$GROUPICON=User.png,$CATICON=User.png*)
	VAR_IN_OUT
		In : BOOL; (*The BOOL var set/reset by the command*)
		Com : INT; (*Command. 1 to set and 0 to reset. After a command, the function sets it to -1*)
	END_VAR
END_FUNCTION

FUNCTION SAFE_UINTDIFF : UINT (*Return the diff of the values of a counte. Takes care about the overflow of the value*) (*$GROUP=User,$CAT=User,$GROUPICON=User.png,$CATICON=User.png*)
	VAR_INPUT
		uiLastValue : UINT;
		uiPrevValue : UINT;
	END_VAR
END_FUNCTION

FUNCTION DintTransfer : BOOL (*Return the value of and DINT splitted in 2 INT values*) (*$GROUP=User,$CAT=User,$GROUPICON=User.png,$CATICON=User.png*)
	VAR_INPUT
		In : DINT; (*DINT to split*)
	END_VAR
	VAR_IN_OUT
		LSint : INT; (*Less significant INT*)
		MSint : INT; (*Most significant INT*)
	END_VAR
END_FUNCTION

FUNCTION StatusAnalogInput : BOOL (*TODO: Add your comment here*) (*$GROUP=User,$CAT=User,$GROUPICON=User.png,$CATICON=User.png*)
	VAR_INPUT
		xModuleOK : BOOL;
		iStatus01 : USINT;
		iStatus02 : USINT;
		iInputNumber : USINT;
	END_VAR
	VAR
		iStatusInput : USINT;
	END_VAR
END_FUNCTION

FUNCTION StatusTemperatureInput : BOOL (*TODO: Add your comment here*) (*$GROUP=User,$CAT=User,$GROUPICON=User.png,$CATICON=User.png*)
	VAR_INPUT
		iStatusTempInput01 : USINT;
		iTemperatureInputNumber : USINT;
	END_VAR
	VAR
		iStatusTemperatureInput : USINT;
	END_VAR
END_FUNCTION

FUNCTION StatusAnalogInputBroken : BOOL (*TODO: Add your comment here*) (*$GROUP=Functions,$CAT=User,$GROUPICON=User.png,$CATICON=User.png*)
	VAR_INPUT
		xModuleOK : BOOL;
		iStatus01 : USINT;
		iStatus02 : USINT;
		iInputNumber : USINT;
	END_VAR
	VAR
		iStatusInput : USINT;
	END_VAR
END_FUNCTION

{REDUND_ERROR} FUNCTION UDINTFromComms : UDINT (*Assignation of a UDINT Double value from an array*) (*$GROUP=User,$CAT=User,$GROUPICON=User.png,$CATICON=User.png*)
	VAR_INPUT
		indexLSB : UINT;
		comsArray : REFERENCE TO ARRAY[0..9999] OF INT;
	END_VAR
END_FUNCTION

{REDUND_ERROR} FUNCTION UDINTToComms : BOOL (*Insert a UDINT value in an array for comms*) (*$GROUP=User,$CAT=User,$GROUPICON=User.png,$CATICON=User.png*)
	VAR_INPUT
		value : UDINT;
		indexLSB : UINT;
		comsArray : REFERENCE TO ARRAY[0..9999] OF INT;
	END_VAR
END_FUNCTION

{REDUND_ERROR} FUNCTION Mmin_TO_DriveUnitsRatio : REAL (*TODO: Add your comment here*) (*$GROUP=User,$CAT=User,$GROUPICON=User.png,$CATICON=User.png*)
	VAR_INPUT
		rDiameter : REAL; (*Value in mm*)
		rGearBox : REAL; (*GearBox ratio (x:1)*)
		rUnitsPerTurn : REAL; (*Units per turn*)
	END_VAR
END_FUNCTION

FUNCTION UINT_SUB : UINT (*UINT substraction. If the result in negative, returns a Cero*)
	VAR_INPUT
		Minuend : UINT; (*Minuend of the substraction*)
		Subtrahend : UINT; (*Subtrahend of the substration*)
	END_VAR
END_FUNCTION

FUNCTION UDINT_SUB : UDINT (*UINT substraction. If the result in negative, returns a Cero*)
	VAR_INPUT
		Minuend : UDINT; (*Minuend of the substraction*)
		Subtrahend : UDINT; (*Subtrahend of the substration*)
	END_VAR
END_FUNCTION

FUNCTION LoadPIDparam : BOOL (*Load the data of the USER structure stPIDParam into the FB structure MTPIDParametersType. VOID*)
	VAR_INPUT
		FB_Structure : REFERENCE TO MTPIDParametersType; (*Structure of the FunctionBlock*)
		USER_Structure : REFERENCE TO stPIDParam; (*Structure of the USER*)
	END_VAR
END_FUNCTION

FUNCTION PLC_Init : BOOL (*Load initial script for PLC. VOID*)
	VAR_INPUT
		plcStruct : REFERENCE TO StPLC; (*StPLC structure*)
	END_VAR
	VAR
		strAux : STRING[80];
	END_VAR
END_FUNCTION

FUNCTION ShiftArrayForward : UINT (*Shift the values of the array some positions forward. Protected to not go beyond the array*)
	VAR_INPUT
		pArray : UDINT; (*Address of the array. Calling as ADR(myArray)*)
		ArraySize : UDINT; (*Address of the array. Calling as SIZEOF(myArray)*)
		ElementSize : UDINT; (*Address of the array. Calling as SIZEOF(myArray[0])*)
		DestinationPosition : UDINT; (*Position where to move the first element of the array*)
		ElementsToMove : UDINT; (*Quantity of elements to move the array*)
	END_VAR
	VAR
		ElementsInArray : UDINT; (*Size of memory to move*)
	END_VAR
END_FUNCTION

FUNCTION ShiftArrayBackward : UINT (*Shift the values of the array some positions backwards. Protected to not go beyond the array*)
	VAR_INPUT
		pArray : UDINT; (*Address of the array. Calling as ADR(myArray)*)
		ArraySize : UDINT; (*Address of the array. Calling as SIZEOF(myArray)*)
		ElementSize : UDINT; (*Address of the array. Calling as SIZEOF(myArray[0])*)
		SourcePosition : UDINT; (*Position to be moved to the first element of the array*)
		ElementsToMove : UDINT; (*Quantity of elements to move the array*)
	END_VAR
	VAR
		ElementsInArray : UDINT; (*Size of memory to move*)
	END_VAR
END_FUNCTION

FUNCTION ShiftArrayOffset : UINT (*Shift the values of the array some positions forward. Protected to not go beyond the array*)
	VAR_INPUT
		pArray : UDINT; (*Address of the array. Calling as ADR(myArray)*)
		ArraySize : UDINT; (*Address of the array. Calling as SIZEOF(myArray)*)
		ElementSize : UDINT; (*Address of the array. Calling as SIZEOF(myArray[0])*)
		SourcePosition : UDINT; (*Position where to move the first element of the array*)
		DestinationPosition : UDINT; (*Position where to move the first element of the array*)
		ElementsToMove : UDINT; (*Quantity of elements to move the array*)
	END_VAR
	VAR
		ElementsInArray : UDINT; (*Size of memory to move*)
	END_VAR
END_FUNCTION

FUNCTION CleanEndArray : UINT (*Write 0 to end of an array to clean of not considered values. Protected to not go beyond the array*)
	VAR_INPUT
		pArray : UDINT; (*Address of the array. Calling as ADR(myArray)*)
		ArraySize : UDINT; (*Address of the array. Calling as SIZEOF(myArray)*)
		ElementSize : UDINT; (*Address of the array. Calling as SIZEOF(myArray[0])*)
		TotalElements : UDINT; (*Position where to move the first element of the array*)
	END_VAR
	VAR
		ElementsToClean : UDINT; (*Quantity of elements to move the array*)
		MaxElementsInArray : UDINT; (*Size of memory to move*)
	END_VAR
END_FUNCTION

FUNCTION TimeFromMmAndMmin : TIME (*Time in ms to run a distance in mm with speed in m/min*)
	VAR_INPUT
		rDistance : REAL; (*Distance in mm*)
		rSpeed : REAL; (*Speed in m/min*)
	END_VAR
END_FUNCTION
```

#### ComandBool.st - Command bool
```iecst
(* TODO: Add your comment here *)
FUNCTION ComandBoolReset

	IF Com = 1 THEN
		In := FALSE;
	END_IF

	Com := -1;
	ComandBoolReset := In;

END_FUNCTION
```

#### ComandBoolReset.st - Command bool
```iecst
(* TODO: Add your comment here *)
FUNCTION ComandBool

	IF Com = 1 THEN
		In := TRUE;
	END_IF

	IF Com = 0 THEN
		In := FALSE;
	END_IF

	Com := -1;
	ComandBool := In;
END_FUNCTION
```

#### SAFE_UINTDIFF.st
```iecst
(* TODO: Add your comment here *)
FUNCTION SAFE_UINTDIFF
	IF uiLastValue >= uiPrevValue THEN
		SAFE_UINTDIFF:= uiLastValue - uiPrevValue;
	ELSE
		SAFE_UINTDIFF:= 65535 - uiPrevValue  + uiLastValue + 1;
	END_IF

(*
	IF data.signals.in.iTachNegative > uiNegTachoCounterPrev THEN
		iDiffPulseTachoNeg:= data.signals.in.iTachNegative - uiNegTachoCounterPrev;
	ELSE
		iDiffPulseTachoNeg:= 65535 + data.signals.in.iTachNegative - uiNegTachoCounterPrev;
	END_IF
*)
END_FUNCTION
```

#### StatusAnalogInput.st - Status analog inputs
```iecst
// Analog Input state
FUNCTION StatusAnalogInput

	//If Module is NOT OK, directly It returns an error in the input, xVacuum1SensorError or xVacuum2SensorError
	IF NOT xModuleOK THEN
		StatusAnalogInput:=TRUE;
		RETURN;
	END_IF

	//Channels 1 to 4 in StatusInput01
	IF iInputNumber>=1 AND iInputNumber<=4 THEN
		iStatusInput:= SHR(iStatus01,(iInputNumber-1)*2) AND 16#03;
	END_IF

	//Channels 5 to 8 in StatusInput02
	IF iInputNumber>=5 AND iInputNumber<=8 THEN
		iStatusInput:= SHR(iStatus02,(iInputNumber-5)*2) AND 16#03;
	END_IF

	StatusAnalogInput:= iStatusInput > 0;

END_FUNCTION
```

#### StatusAnalogInputBroken.st
```iecst
// Analog Input state
FUNCTION StatusAnalogInputBroken

	//If Module is NOT OK, directly It returns an error in the input, xVacuum1SensorError or xVacuum2SensorError
	IF NOT xModuleOK THEN
		StatusAnalogInputBroken:=TRUE;
		RETURN;
	END_IF

	//Channels 1 to 4 in StatusInput01
	IF iInputNumber>=1 AND iInputNumber<=4 THEN
		iStatusInput:= SHR(iStatus01,(iInputNumber-1)*2) AND 16#01;
	END_IF

	//Channels 5 to 8 in StatusInput02
	IF iInputNumber>=5 AND iInputNumber<=8 THEN
		iStatusInput:= SHR(iStatus02,(iInputNumber-5)*2) AND 16#01;
	END_IF

	StatusAnalogInputBroken:= iStatusInput > 0;

END_FUNCTION
```

#### UDINT_SUB.st
```iecst
(* TODO: Add your comment here *)
FUNCTION UDINT_SUB

	//Protection of values to avoid infinite values
	IF Minuend >= Subtrahend THEN
		UDINT_SUB := Minuend - Subtrahend;
	ELSE
		UDINT_SUB := 0;
	END_IF

END_FUNCTION
```

#### LoadPIDparam.st
```iecst
(* TODO: Add your comment here *)
FUNCTION LoadPIDparam

	FB_Structure.Gain 				:= USER_Structure.rKp;
	FB_Structure.IntegrationTime	:= USER_Structure.rTi;
	FB_Structure.DerivativeTime 	:= USER_Structure.rKd;
	FB_Structure.FilterTime 		:= USER_Structure.rTd;

	LoadPIDparam := TRUE;

END_FUNCTION
```

#### Arrays.st
```iecst
(* Shift the values of the array some positions forward. Protected to not go beyond the array. UINT *)
FUNCTION ShiftArrayForward

	ShiftArrayForward := ShiftArrayOffset(pArray, ArraySize, ElementSize, 0, DestinationPosition, ElementsToMove);

END_FUNCTION

(* Shift the values of the array some positions forward. Protected to not go beyond the array. UINT *)
FUNCTION ShiftArrayBackward

(* ------ List of possible status ---------------------
	0:		Shift OK
	1:		Shift Done but limited
	50000:	Zero elements to move selected
	50001:	Source position outside array bounds
	50002:	Array pointer not assigned
-------------------------------------------------------*)

    //Check if an element has to be moved - If not status 50000 is reported
	IF ElementsToMove = 0 THEN
		ShiftArrayBackward := 50000;
		RETURN;
	END_IF

	//Check if the source position is in the array boundaries - If not status 50001 is reported
	ElementsInArray := ArraySize / ElementSize;
	IF SourcePosition >= ElementsInArray THEN
		ShiftArrayBackward := 50001;
		RETURN;
	END_IF

	// Check if pointer of array is assigned
	IF pArray = 0 THEN
		ShiftArrayBackward := 50002;
		RETURN;
	END_IF

	//Check if the movement goes outside the array and limit it to the maximum size of the array - Status 0 is reported

	IF ElementsInArray - SourcePosition < ElementsToMove THEN
		brsmemmove(pArray, pArray+ElementSize*SourcePosition, (ElementsInArray-SourcePosition)*ElementSize);
		ShiftArrayBackward := 1;
	ELSE
		brsmemmove(pArray, pArray+ElementSize*SourcePosition, ElementsToMove*ElementSize);
		ShiftArrayBackward := 0;
	END_IF

END_FUNCTION

(* Shift the values of the array some positions forward. Protected to not go beyond the array. UINT *)
FUNCTION ShiftArrayOffset

(* ------ List of possible status ---------------------
	0:		Shift OK
	1:		Shift Done but limited
	50000:	Zero elements to move selected
	50001:	Destination position outside array bounds
	50002:	Array pointer not assigned
	50003:	Source and destination are the same
-------------------------------------------------------*)

    //Check if an element has to be moved - If not status 50000 is reported
	IF ElementsToMove = 0 THEN
		ShiftArrayOffset := 50000;
		RETURN;
	END_IF

	//Check if the destination position is in the array boundaries - If not status 50001 is reported
	ElementsInArray := ArraySize / ElementSize;
	IF DestinationPosition >= ElementsInArray THEN
		ShiftArrayOffset := 50001;
		RETURN;
	END_IF

	// Check if pointer of array is assigned
	IF pArray = 0 THEN
		ShiftArrayOffset := 50002;
		RETURN;
	END_IF

	// Check if source and Destination position
	IF SourcePosition = DestinationPosition THEN
		ShiftArrayOffset := 50003;
		RETURN;
	END_IF

	//Check if the movement goes outside the array and limit it to the maximum size of the array - Status 0 is reported
	IF ElementsInArray - DestinationPosition < ElementsToMove THEN
		brsmemmove(pArray+ElementSize*DestinationPosition, pArray+ElementSize*SourcePosition, (ElementsInArray-DestinationPosition)*ElementSize);
		ShiftArrayOffset := 1;
	ELSE
		brsmemmove(pArray+ElementSize*DestinationPosition, pArray+ElementSize*SourcePosition, ElementsToMove*ElementSize);
		ShiftArrayOffset := 0;
	END_IF

END_FUNCTION

(* Shift the values of the array some positions forward. Protected to not go beyond the array. UINT *)
FUNCTION CleanEndArray

(* ------ List of possible status ---------------------
	0:		Clean OK
	1:		Shift Done but limited
	//50000:	Zero elements to move selected
	50001:	Total elements greater than the maximum allowed
	50002:	Array pointer not assigned
	50003:	No space at the end of the array
-------------------------------------------------------*)

	// Check if pointer of array is assigned
	IF pArray = 0 THEN
		CleanEndArray := 50002;
		RETURN;
	END_IF

	// If no elements, clean all the array
	IF TotalElements = 0 THEN
		brsmemset(pArray, 0, ArraySize);
		CleanEndArray := 0;
		RETURN;
	END_IF

	//Check if the destination position is in the array boundaries - If not status 50001 is reported
	MaxElementsInArray := ArraySize / ElementSize;
	IF TotalElements > MaxElementsInArray THEN
		CleanEndArray := 50001;
		RETURN;
	END_IF

	ElementsToClean := MaxElementsInArray - TotalElements;

	// If the elements is the same as the maximum, no space to clean
	IF ElementsToClean = 0 THEN
		CleanEndArray := 50003;
		RETURN;
	END_IF

	brsmemset(pArray + ElementSize*TotalElements, 0, ElementSize*ElementsToClean);
	CleanEndArray := 0;

END_FUNCTION
```

### Library Logical/ExtPack/EFILib/EFILib_v1/ConvertFun (IEC) - Conversion data functions

#### ConvertFun.fun - Exported functions and function blocks
```iecst
FUNCTION SECONDS_TO_MILLIS : UDINT (*TODO: Add your comment here*) (*$GROUP=User,$CAT=User,$GROUPICON=User.png,$CATICON=User.png*)
	VAR_INPUT
		iSeconds : UDINT;
	END_VAR
END_FUNCTION

FUNCTION MINUTES_TO_MILLIS : UDINT (*TODO: Add your comment here*) (*$GROUP=User,$CAT=User,$GROUPICON=User.png,$CATICON=User.png*)
	VAR_INPUT
		minutes : UINT;
	END_VAR
END_FUNCTION

FUNCTION MILLISECONDS_TO_TIME : TIME
	VAR_INPUT
		iMilliSeconds : UDINT;
	END_VAR
END_FUNCTION

FUNCTION SECONDS_TO_TIME : TIME
	VAR_INPUT
		iSeconds : UDINT;
	END_VAR
END_FUNCTION

FUNCTION MINUTES_TO_TIME : TIME
	VAR_INPUT
		iMinutes : UINT;
	END_VAR
END_FUNCTION

FUNCTION TIME_TO_MINUTES : UINT
	VAR_INPUT
		tiTimeValue : TIME;
	END_VAR
END_FUNCTION

FUNCTION TIME_TO_SECONDS : UDINT
	VAR_INPUT
		tiTimeValue : TIME;
	END_VAR
END_FUNCTION

FUNCTION TIME_TO_SECONDS_COMS : UINT
	VAR_INPUT
		tiTimeValue : TIME;
	END_VAR
END_FUNCTION

FUNCTION TIME_TO_MILLISECONDS : UDINT
	VAR_INPUT
		tiTimeValue : TIME;
	END_VAR
END_FUNCTION

FUNCTION TIME_TO_MILLISECONDS_COMS : UINT
	VAR_INPUT
		tiTimeValue : TIME;
	END_VAR
END_FUNCTION
```

#### MINUTES_TO_MILLIS.st
```iecst
(* TODO: Add your comment here *)
FUNCTION MINUTES_TO_MILLIS
	MINUTES_TO_MILLIS := minutes*60*1000;
END_FUNCTION
```

#### MILLISECONDS_TO_TIME.st
```iecst
(* TODO: Add your comment here *)
FUNCTION MILLISECONDS_TO_TIME

	MILLISECONDS_TO_TIME := UDINT_TO_TIME(iMilliSeconds);

END_FUNCTION
```

#### MINUTES_TO_TIME.st
```iecst
(* TODO: Add your comment here *)
FUNCTION MINUTES_TO_TIME

	MINUTES_TO_TIME := UDINT_TO_TIME(MINUTES_TO_MILLIS(iMinutes));	//Time conversion needs

END_FUNCTION
```

### Package Logical/ExtPack/_Motion/AxisCtrl - Axis Ctrl Logic package

### Package Logical/ExtPack/_Motion/AxisCtrl/AxisCtrl_v2 - Axis Ctrl Logic package. Gear inside AxisCtrl

### Program Logical/ExtPack/_Motion/AxisCtrl/AxisCtrl_v2/AxisCtrl

#### AxisCtrl.var
```iecst
(********************************************************************
 * COPYRIGHT - B&R Spain
 ********************************************************************
 * Program: AxisCtrl
 * File: AxisCtrl.var
 * Author: B&R Spain
 * Created: September 19, 2013
 ********************************************************************
 * Local variables of program AxisCtrl
 ********************************************************************)
(********************************************************************
 * Configuration of StateSupervisor
********************************************************************)
VAR CONSTANT
	TIMEOUT_SWITCH_ON_OFF : TIME := T#10s; (*Maximum time that the axis is allowed to wait for switch on or off. It must be at least 7s in order to be able to get the 4005 error*)
	TIMEOUT_STATE_EXCEPTION : TIME := T#500ms; (*Maximum time that the axis is allowed to have an unexpected state*)
END_VAR
(********************************************************************
 * References
********************************************************************)
VAR
	AdrEncoderData : UDINT; (*Address of the permanent variable where the encoder data is stored*)
	pAxisCtrl : REFERENCE TO AxisCtrl_typ; (*Axis control structure (local reference to avoid doing a find & replace)*)
	isqRippleData : REFERENCE TO MC_ISQ_RippleData_typ;
	AxisRef : UDINT; (*Axis reference (address of ACP10 structure)*)
	MasterRef : UDINT; (*Axis reference (address of ACP10 structure)*)
	AxisName : STRING[12];
	MasterName : STRING[12];
END_VAR
(********************************************************************
 * Sequences
********************************************************************)
VAR
	InitStep : USINT; (*Current step in the init step sequence*)
	AxisState : AxisState_typ; (*Current step in the step sequence*)
	AxisErrorState : AxisErrorState_typ; (*Current step in the error handling step sequence*)
END_VAR
(********************************************************************
 * FBKs
********************************************************************)
VAR
	MC_ReadStatus_0 : MC_ReadStatus; (*Function Block*)
	MC_BR_ReadDriveStatus_0 : MC_BR_ReadDriveStatus; (*Function Block*)
	MC_ReadAxisError_0 : MC_ReadAxisError; (*Function Block*)
	MC_ReadActualPosition_0 : MC_ReadActualPosition; (*Function Block *)
	MC_ReadActualVelocity_0 : MC_ReadActualVelocity; (*Function Block*)
	MC_ReadActualTorque_0 : MC_ReadActualTorque; (*Function Block *)
	MC_Power_0 : MC_Power; (*Function Block*)
	MC_Home_0 : MC_Home; (*Function Block*)
	MC_MoveAbsolute_0 : MC_MoveAbsolute; (*Function Block*)
	MC_MoveAbsolute_1 : MC_MoveAbsolute; (*Function Block*)
	MC_MoveAdditive_0 : MC_MoveAdditive; (*Function Block*)
	MC_MoveAdditive_1 : MC_MoveAdditive; (*Function Block*)
	MC_MoveVelocity_0 : MC_MoveVelocity; (*Function Block*)
	MC_MoveVelocity_1 : MC_MoveVelocity; (*Function Block*)
	MC_GearIn_0 : MC_GearIn; (*Function Block*)
	MC_GearIn_1 : MC_GearIn; (*Function Block*)
	MC_GearOut_x : MC_GearOut; (*Function Block*)
	MC_Halt_0 : MC_Halt; (*Function Block*)
	MC_Halt_1 : MC_Halt; (*Function Block*)
	MC_Stop_0 : MC_Stop; (*Function Block*)
	MC_Reset_0 : MC_Reset; (*Function Block*)
	MC_SetOverride_0 : MC_SetOverride; (*Function Block*)
	MC_BR_InitEndlessPosition_0 : MC_BR_InitEndlessPosition; (*Function Block*)
	MC_ReadMotorTemp : MC_BR_CyclicRead;
	MC_ReadAmbTemp : MC_BR_ReadParID;
	MC_BR_WriteParIDText_EncReset : MC_BR_WriteParIDText; (*Function Block*)
END_VAR
(********************************************************************
 * Temp Variables
********************************************************************)
VAR
	StatusNcAccess : UINT;
	AxisRefDone : BOOL;
	pACP10VAXIS : REFERENCE TO ACP10VAXIS_typ;
	pACP10AXIS : REFERENCE TO ACP10AXIS_typ;
	AxisIsVirtual : BOOL;
	MasterRefDone : BOOL;
	InitDone : BOOL;
	InPosition : BOOL;
	InGear : BOOL;
	HomeValid : BOOL;
	ErrorTextFB : ARRAY[0..3] OF STRING[79];
	DriveStatusFB : MC_DRIVESTATUS_TYP;
	InitErrorText : ARRAY[0..3] OF STRING[79];
	InitErrorID : UINT;
	InitErrorSource : AxisCtrl_errorSource_enu;
	ErrorText : ARRAY[0..3] OF STRING[79];
	ErrorAux : STRING[79];
	ErrorFB : STRING[79];
	ErrorID : UINT;
	ErrorSource : AxisCtrl_errorSource_enu;
	TON_Exception : TON;
	R_TRIG_JogStepByStepPos : R_TRIG;
	R_TRIG_JogStepByStepNeg : R_TRIG;
	iActualCommandsCounter : USINT;
	MC_BR_WriteParID_31 : MC_BR_WriteParID;
	MC_BR_ReadParID_11 : MC_BR_ReadParID; (*Read Max Temperature of Drivers*)
	MC_BR_CyclicRead_10 : MC_BR_ReadParID; (*Read Actual Temperature of Driver*)
	MC_BR_CyclicRead_20 : MC_BR_ReadParID; (*Read Actual Temperature of Motors*)
	MC_BR_ReadParID_51 : MC_BR_ReadParID; (*Read Max speed of Motors*)
	MC_BR_ReadParID_21 : MC_BR_ReadParID; (*Read Max Temperature of Motors*)
	MC_BR_ReadParID_913 : MC_BR_ReadParID;
	MC_BR_ReadParID_914 : MC_BR_ReadParID;
	MC_BR_ReadParID_915 : MC_BR_ReadParID;
	MC_BR_ReadParID_916 : MC_BR_ReadParID;
	MC_BR_WriteParID_30 : MC_BR_WriteParID;
	MC_BR_WriteParID_32 : MC_BR_WriteParID;
	MC_BR_WriteParID_33 : MC_BR_WriteParID;
	MC_BR_WriteParID_34 : MC_BR_WriteParID;
	MC_BR_WriteParID_35 : MC_BR_WriteParID;
	MC_BR_WriteParID_36 : MC_BR_WriteParID;
	MC_BR_WriteParID_37 : MC_BR_WriteParID;
	MC_BR_WriteParID_38 : MC_BR_WriteParID;
	MC_BR_WriteParID_39 : MC_BR_WriteParID;
	MC_BR_WriteParID_40 : MC_BR_WriteParID;
	MC_BR_WriteParID_41 : MC_BR_WriteParID;
	MC_BR_WriteParID_42 : MC_BR_WriteParID;
	MC_BR_WriteParID_43 : MC_BR_WriteParID;
	MC_BR_WriteParID_44 : MC_BR_WriteParID;
	MC_BR_WriteParID_45 : MC_BR_WriteParID;
	MC_BR_ReadParID_112 : MC_BR_ReadParID; (*To read param Id acceleration*)
	MC_BR_ReadParID_214 : MC_BR_ReadParID; (*To read param Id acceleration*)
	MC_BR_ReadParID_53 : MC_BR_ReadParID; (*To read param Id acceleration*)
	MC_BR_ReadParID_54 : MC_BR_ReadParID; (*To read param Id acceleration*)
	PowerStatusOld : BOOL; (*MC_BR_WriteParID_0 : MC_BR_WriteParID;
	MC_BR_WriteParID_1 : MC_BR_WriteParID;
	MC_BR_WriteParID_2 : MC_BR_WriteParID;
	MC_BR_WriteParID_3 : MC_BR_WriteParID;
	MC_BR_WriteParID_4 : MC_BR_WriteParID;
	MC_BR_WriteParID_5 : MC_BR_WriteParID;
	MC_BR_WriteParID_6 : MC_BR_WriteParID;
	MC_BR_WriteParID_7 : MC_BR_WriteParID;
	MC_BR_WriteParID_8 : MC_BR_WriteParID;
	MC_BR_WriteParID_9 : MC_BR_WriteParID;
	MC_BR_WriteParID_10 : MC_BR_WriteParID;
	MC_BR_WriteParID_11 : MC_BR_WriteParID;
	MC_BR_WriteParID_14 : MC_BR_WriteParID;
	MC_BR_WriteParID_15 : MC_BR_WriteParID;*)
	MasterUsed : BOOL; (*Master-Slave Function is Used in Axis Control*)
END_VAR
(********************************************************************
 * ISQ RIPPLE Variables
********************************************************************)
VAR
	isqRippleDataEmpty : MC_ISQ_RippleData_typ;
	urISQdataValue : REAL;
	udiISQdataValue : UDINT;
	udiISQdataAddres : UDINT;
	uiISQparId : UINT;
	iISQTimesInReadUpload : USINT;
	iISQTimesInWriteUpload : USINT;
	xISQOrderWriteUploadCount : UINT;
	xISQOrderWriteUpload : BOOL;
	xISQOrderReadUploadCount : UINT;
	xISQOrderReadUpload : BOOL;
	fbISQWriteParUpload : MC_BR_WriteParID;
	fbISQReadParUpload : MC_BR_ReadParID;
	iISQUploadindex : USINT := 100; (*This value to 90 is the start order*)
	iISQUploadsubindex : USINT := 100;
	xISQUploadnext : BOOL := FALSE;
	iISQTimesInReadDownload : USINT;
	iISQTimesInWriteDownload : USINT;
	xISQOrderWriteDownloadCount : UINT;
	xISQOrderWriteDownload : BOOL;
	xISQOrderWriteSingleDownloadCnt : UINT;
	xISQOrderWriteSingleDownload : BOOL;
	fbISQWriteParDownload : MC_BR_WriteParID;
	fbISQWriteSingleParDownload : MC_BR_WriteParID;
	iISQDownloadindex : USINT := 100; (*This value to 90 is the start order*)
	iISQDownloadsubindex : USINT := 100;
	xISQDownloadnext : BOOL := FALSE;
	iCommandsError : DINT;
	rActualCurrent : REAL; (*Value to assign the reading of the FB*)
END_VAR
```

#### InitSequence.st
```iecst
(********************************************************************
 * COPYRIGHT - B&R Spain
 ********************************************************************
 * PROGRAM: AxisCtrlTRUE
 * File: InitSequence.st
 * Author: B&R Spain
 * Created: September 19, 2013
 * Modified: February 17, 2016
 ********************************************************************
 * Implementation of action InitSequence
 ********************************************************************)

ACTION InitSequence:

	IF EDGEPOS( NOT DriveStatusFB.NetworkInit) THEN
		InitStep := 0;
		InitDone := FALSE;
		MC_BR_WriteParID_30(Axis := AxisRef, Execute := FALSE);
		MC_BR_WriteParID_31(Axis := AxisRef, Execute := FALSE);
		MC_BR_WriteParID_32(Axis := AxisRef, Execute := FALSE);
		MC_BR_WriteParID_33(Axis := AxisRef, Execute := FALSE);
		MC_BR_WriteParID_34(Axis := AxisRef, Execute := FALSE);
		MC_BR_WriteParID_35(Axis := AxisRef, Execute := FALSE);
		MC_BR_WriteParID_36(Axis := AxisRef, Execute := FALSE);
		MC_BR_WriteParID_37(Axis := AxisRef, Execute := FALSE);
		MC_BR_WriteParID_38(Axis := AxisRef, Execute := FALSE);
		MC_BR_WriteParID_39(Axis := AxisRef, Execute := FALSE);
		MC_BR_WriteParID_40(Axis := AxisRef, Execute := FALSE);
		MC_BR_WriteParID_41(Axis := AxisRef, Execute := FALSE);
		MC_BR_WriteParID_42(Axis := AxisRef, Execute := FALSE);
		MC_BR_WriteParID_43(Axis := AxisRef, Execute := FALSE);
		MC_BR_WriteParID_44(Axis := AxisRef, Execute := FALSE);
		MC_BR_WriteParID_45(Axis := AxisRef, Execute := FALSE);
	END_IF;

    CASE InitStep OF

        0: (* Set default parameters *)

			pAxisCtrl.Parameter.Override.Speed           := 1.0;    		(* multiplication factor for override velocity *)
			pAxisCtrl.Parameter.Override.Acceleration    := 1.0;     		(* multiplication factor for override acceleration *)

            InitStep := 10;

        10: (* Get ACP10 axis reference *)

			//StatusNcAccess := ncaccess(ncACP10MAN, ADR(AxisName), ADR(AxisRef));  //This is the original code
			AxisName:=pAxisCtrl.Parameter.Init.AxisObjectName;
			StatusNcAccess := ncaccess(ncACP10MAN, ADR(AxisName), ADR(AxisRef));
            IF StatusNcAccess = 0 THEN
                AxisRefDone := TRUE;
                InitErrorID := 0;
                InitErrorSource := ERR_SRC_NO_ERROR;
                InitErrorText[0] := '';
                InitErrorText[1] := '';
                InitStep := 11;
            ELSE
                InitErrorID := 29200;
                InitErrorSource := ERR_SRC_TASK;
                InitErrorText[0] := 'The axis object is invalid';
                InitErrorText[1] := 'AxisName in the References.st file must match the one in the NC mapping';
            END_IF

        11: (* Determine if axis is real or virtual *)

            pACP10AXIS ACCESS AxisRef;
            pACP10VAXIS ACCESS AxisRef;
            IF pACP10AXIS.nc_obj_inf.nc_obj_typ = ncAXIS THEN
                AxisIsVirtual := FALSE;
            ELSIF pACP10VAXIS.nc_obj_inf.nc_obj_typ = ncV_AXIS THEN
                AxisIsVirtual := TRUE;
            END_IF
			InitStep := 12;

		12: (* Get ACP10 master axis reference *)

			MasterName:=pAxisCtrl.Parameter.Init.MasterGearObjectName;
			IF MasterName <> '' THEN
				StatusNcAccess := ncaccess(ncACP10MAN, ADR(MasterName), ADR(MasterRef));
				MasterUsed := TRUE;
				IF StatusNcAccess = 0 THEN
					MasterRefDone := TRUE;
					InitErrorID := 0;
					InitErrorSource := ERR_SRC_NO_ERROR;
					InitErrorText[0] := '';
					InitErrorText[1] := '';
					InitStep := 20;
				ELSE
					InitErrorID := 29200;
					InitErrorSource := ERR_SRC_TASK;
					InitErrorText[0] := 'The axis object is invalid';
					InitErrorText[1] := 'MasterName in the References.st file must match the one in the NC mapping';
				END_IF
			ELSE (* If master axis is not specified, the EngageToMaster command will not be available *)
				MasterUsed := FALSE;
				InitStep := 20;
			END_IF

        20: (* Init endless position (for MC_HOME_RESTORE_POS mode) *)

            IF AdrEncoderData <> 0 THEN
                IF MC_ReadStatus_0.Disabled OR MC_ReadStatus_0.StandStill THEN
                    MC_BR_InitEndlessPosition_0.Execute := TRUE;
                    MC_BR_InitEndlessPosition_0.DataAddress := AdrEncoderData;
                    InitStep := 21;
                END_IF
            ELSIF DriveStatusFB.NetworkInit THEN (* If the address is not specified, the step is skipped and the MC_HOME_RESTORE_POS is not available *)
                InitStep := 30;
            END_IF
        21:
            IF MC_BR_InitEndlessPosition_0.Done THEN
                MC_BR_InitEndlessPosition_0.Execute := FALSE;
                InitStep := 30;
            END_IF
            IF MC_BR_InitEndlessPosition_0.Error THEN
                MC_BR_InitEndlessPosition_0.Execute := FALSE;
                InitStep := 20;
            END_IF

			// ########################### SEND VELOCITY PARAMETERS ###########################
		30:
			IF pAxisCtrl.Parameter.Init.xSendVelParams THEN

				MC_BR_WriteParID_30(Axis := AxisRef, Execute := TRUE, ParID := ACP10PAR_AXLIM_V_POS, DataAddress := ADR(pAxisCtrl.Parameter.Init.rLimitVelPos), DataType := ncPAR_TYP_REAL);
				IF MC_BR_WriteParID_30.Done THEN
					InitStep := 31;
				END_IF

			ELSE
				InitStep := 31;
			END_IF

		31:
			IF pAxisCtrl.Parameter.Init.xSendVelParams THEN

				MC_BR_WriteParID_31(Axis := AxisRef, Execute := TRUE, ParID := ACP10PAR_AXLIM_V_NEG, DataAddress := ADR(pAxisCtrl.Parameter.Init.rLimitVelNeg), DataType := ncPAR_TYP_REAL);

				IF MC_BR_WriteParID_31.Done THEN
					InitStep := 32;
				END_IF

			ELSE
				InitStep := 32;
			END_IF

		// ########################### SEND ACCELERATION PARAMETERS ###########################
		32:
			IF pAxisCtrl.Parameter.Init.xSendAccParams THEN

				MC_BR_WriteParID_32(Axis := AxisRef, Execute := TRUE, ParID := ACP10PAR_AXLIM_A1_POS, DataAddress := ADR(pAxisCtrl.Parameter.Init.rLimitAccPos), DataType := ncPAR_TYP_REAL);

				IF MC_BR_WriteParID_32.Done THEN
					InitStep := 33;
				END_IF
			ELSE
				InitStep := 33;
			END_IF

		33:
			IF pAxisCtrl.Parameter.Init.xSendAccParams THEN

				MC_BR_WriteParID_33(Axis := AxisRef, Execute := TRUE, ParID := ACP10PAR_AXLIM_A2_POS, DataAddress := ADR(pAxisCtrl.Parameter.Init.rLimitAccPos), DataType := ncPAR_TYP_REAL);

				IF MC_BR_WriteParID_33.Done THEN
					InitStep := 34;
				END_IF

			ELSE
				InitStep := 34;
			END_IF

		34:
			IF pAxisCtrl.Parameter.Init.xSendAccParams THEN

				MC_BR_WriteParID_34(Axis := AxisRef, Execute := TRUE, ParID := ACP10PAR_AXLIM_A1_NEG, DataAddress := ADR(pAxisCtrl.Parameter.Init.rLimitAccNeg), DataType := ncPAR_TYP_REAL);

				IF MC_BR_WriteParID_34.Done THEN
					InitStep := 35;
				END_IF

			ELSE
				InitStep := 35;
			END_IF

		35:
			IF pAxisCtrl.Parameter.Init.xSendAccParams THEN

				MC_BR_WriteParID_35(Axis := AxisRef, Execute := TRUE, ParID := ACP10PAR_AXLIM_A2_NEG, DataAddress := ADR(pAxisCtrl.Parameter.Init.rLimitAccNeg), DataType := ncPAR_TYP_REAL);

				IF MC_BR_WriteParID_35.Done THEN
					InitStep := 36;
				END_IF

			ELSE
				InitStep := 36;
			END_IF

			// ########################### SEND EMERGENCY STOP PARAMETERS ###########################
		36:
			IF pAxisCtrl.Parameter.Init.xSendAccEmergStopParams THEN

				MC_BR_WriteParID_36(Axis := AxisRef, Execute := TRUE, ParID := ACP10PAR_LIM_A_SET_STOP, DataAddress := ADR(pAxisCtrl.Parameter.Init.rLimitAccStop), DataType := ncPAR_TYP_REAL);

				IF MC_BR_WriteParID_36.Done THEN
					InitStep := 37;
				END_IF

			ELSE
				InitStep := 37;
			END_IF

			// ########################### SEND TORQUE PARAMETERS ###########################
		37:
			IF pAxisCtrl.Parameter.Init.xSendTorqueParams THEN

				MC_BR_WriteParID_37(Axis := AxisRef, Execute := TRUE, ParID := ACP10PAR_LIM_T1_POS, DataAddress := ADR(pAxisCtrl.Parameter.Init.rLimitTorquePos), DataType := ncPAR_TYP_REAL);

				IF MC_BR_WriteParID_37.Done THEN
					InitStep := 38;
				END_IF

			ELSE
				InitStep := 38;
			END_IF

		38:
			IF pAxisCtrl.Parameter.Init.xSendTorqueParams THEN

				MC_BR_WriteParID_38(Axis := AxisRef, Execute := TRUE, ParID := ACP10PAR_LIM_T1_NEG, DataAddress := ADR(pAxisCtrl.Parameter.Init.rLimitTorqueNeg), DataType := ncPAR_TYP_REAL);

				IF MC_BR_WriteParID_38.Done THEN
					InitStep := 39;
				END_IF

			ELSE
				InitStep := 39;
			END_IF

		39:
			IF pAxisCtrl.Parameter.Init.xSendTorqueParams THEN

				MC_BR_WriteParID_39(Axis := AxisRef, Execute := TRUE, ParID := ACP10PAR_LIM_T2_POS, DataAddress := ADR(pAxisCtrl.Parameter.Init.rLimitTorquePos), DataType := ncPAR_TYP_REAL);

				IF MC_BR_WriteParID_39.Done THEN
					InitStep := 40;
				END_IF

			ELSE
				InitStep := 40;
			END_IF
		40:
			IF pAxisCtrl.Parameter.Init.xSendSwEndParams THEN

				MC_BR_WriteParID_40(Axis := AxisRef, Execute := TRUE, ParID := ACP10PAR_LIM_T2_NEG, DataAddress := ADR(pAxisCtrl.Parameter.Init.rLimitTorqueNeg), DataType := ncPAR_TYP_REAL);

				IF MC_BR_WriteParID_40.Done THEN
					InitStep := 41;
				END_IF

			ELSE
				InitStep := 41;
			END_IF

			// ########################### SEND SOFWARE END PARAMETERS ###########################
		41:
			IF pAxisCtrl.Parameter.Init.xSendSwEndParams THEN

				MC_BR_WriteParID_41(Axis := AxisRef, Execute := TRUE, ParID := ACP10PAR_AXLIM_POS_SW_END, DataAddress := ADR(pAxisCtrl.Parameter.Init.diLimitPosSwEnd), DataType := ncPAR_TYP_DINT);

				IF MC_BR_WriteParID_41.Done THEN
					InitStep := 42;
				END_IF

			ELSE
				InitStep := 42;
			END_IF

		42:
			IF pAxisCtrl.Parameter.Init.xSendTorqueParams THEN

				MC_BR_WriteParID_42(Axis := AxisRef, Execute := TRUE, ParID := ACP10PAR_AXLIM_NEG_SW_END, DataAddress := ADR(pAxisCtrl.Parameter.Init.diLimitNegSwEnd), DataType := ncPAR_TYP_DINT);

				IF MC_BR_WriteParID_42.Done THEN
					InitStep := 43;
				END_IF

			ELSE
				InitStep := 43;
			END_IF

			// ########################### SEND HOMING PARAMETERS ###########################
		43:
			IF pAxisCtrl.Parameter.Init.xSendHomingParams THEN

				MC_BR_WriteParID_43(Axis := AxisRef, Execute := TRUE, ParID := ACP10PAR_HOMING_V_SWITCH, DataAddress := ADR(pAxisCtrl.Parameter.Init.rHomingVSwitch), DataType := ncPAR_TYP_REAL);

				IF MC_BR_WriteParID_43.Done THEN
					InitStep := 44;
				END_IF

			ELSE
				InitStep := 44;
			END_IF

		44:
			IF pAxisCtrl.Parameter.Init.xSendHomingParams THEN

				MC_BR_WriteParID_44(Axis := AxisRef, Execute := TRUE, ParID := ACP10PAR_HOMING_V_TRIGGER, DataAddress := ADR(pAxisCtrl.Parameter.Init.rHomingVTrigger), DataType := ncPAR_TYP_REAL);

				IF MC_BR_WriteParID_44.Done THEN
					InitStep := 45;
				END_IF

			ELSE
				InitStep := 45;
			END_IF

		45:
			IF pAxisCtrl.Parameter.Init.xSendHomingParams THEN

				MC_BR_WriteParID_45(Axis := AxisRef, Execute := TRUE, ParID := ACP10PAR_HOMING_A, DataAddress := ADR(pAxisCtrl.Parameter.Init.rHomingAcc), DataType := ncPAR_TYP_REAL);

				IF MC_BR_WriteParID_45.Done THEN
					InitStep := 46;
				END_IF

			ELSE
				InitStep := 46;
			END_IF

        46: (* Add here more initialization steps if needed... (e.g. transfer cam to ACOPOS) *)

            (* When all the initializations are done, set the following flag *)
			InitDone := TRUE;

        99: (* Example: transfer a cam profile to the ACOPOS ************************************)
            (* To enable it, do the following steps                                             *)
            (* TODO: Define a cam profile in the Logical View and assign it to the PLC          *)
            (* TODO: Declare the corresponding variables                                        *)
            (* TODO: Add the corresponding FB call at the end OF the cyclic                     *)
            (* TODO: Remember to set the InitDone flag only after all init steps are done       *)
            (*************************************** and add a ')' after the following asterisk *
            MC_BR_DownloadCamProfileObj_0.Execute := TRUE;
            MC_BR_DownloadCamProfileObj_0.DataObjectName := 'CamProfile';
            MC_BR_DownloadCamProfileObj_0.Index := 1;
            MC_BR_DownloadCamProfileObj_0.Periodic := FALSE;
            InitStep := 41;
        41:
            IF MC_BR_DownloadCamProfileObj_0.Done THEN
                MC_BR_DownloadCamProfileObj_0.Execute := FALSE;
                InitStep := 50;
            END_IF
            IF MC_BR_DownloadCamProfileObj_0.Error THEN
                MC_BR_DownloadCamProfileObj_0.Execute := FALSE;
                InitStep := 40;
            END_IF
            (************************************************************************************)

        (************************************************************************************)
        (* In case a minimum or specific ACP10 version would be necessary, this shows how   *)
        (* to detect the ACP10 version from the program:                                    *)
        (* pAxisACP10.sw_version.nc_manager = 16#ABCD <-> ACP10 VA.BC.D                     *)
        (* e.g. 16#2260 <-> V2.26.0                                                         *)
        (* Note that pAxisACP10 must be a pointer to ACP10AXIS_typ or ACP10VAXIS_typ depen- *)
        (* ding on whether the axis is real or virtual.                                     *)
        (************************************************************************************)

    END_CASE

END_ACTION
```

#### StateSupervisor.st
```iecst
(********************************************************************
 * COPYRIGHT - B&R Spain
 ********************************************************************
 * Program: AxisCtrl
 * File: StateSupervisor.st
 * Author: B&R Spain
 * Created: September 19, 2013
 * Modified: April 28, 2017
 ********************************************************************
 * Implementation of action StateSupervisor
 ********************************************************************
 * Whenever an agent outside this program (e.g. the Test Window) or
 * the CNC manager would perform a command that would cause a state
 * change or whenever an unexpected error would occur, this state
 * supervisor would find which is the resulting axis state.
 ********************************************************************)

ACTION StateSupervisor:

    (* Detects exceptions, where axis states are not the expected ones *)
    CASE AxisState OF

        (* States where the PLCopen state must be Disabled *)
        AX_STATE_DISABLED:
            TON_Exception.PT := TIMEOUT_STATE_EXCEPTION;
            (* Virtual axes cannot be in disabled state therefore they are allowed to be in standstill *)
            IF AxisIsVirtual THEN
                TON_Exception.IN := NOT(MC_ReadStatus_0.Disabled OR MC_ReadStatus_0.StandStill);
            ELSE
                TON_Exception.IN := NOT(MC_ReadStatus_0.Disabled);
            END_IF

        AX_STATE_UK_DISABLED:
            TON_Exception.PT := T#0ms;
            (* Virtual axes cannot be in disabled state therefore they are allowed to be in standstill *)
            IF AxisIsVirtual THEN
                TON_Exception.IN := NOT(MC_ReadStatus_0.Disabled OR MC_ReadStatus_0.StandStill);
            ELSE
                TON_Exception.IN := NOT(MC_ReadStatus_0.Disabled);
            END_IF

        (* States where the PLCopen state must be Homing *)
        AX_STATE_HOMING_NO_POWER, AX_STATE_HOMING:
            TON_Exception.PT := TIMEOUT_STATE_EXCEPTION;
            TON_Exception.IN := NOT(MC_ReadStatus_0.Homing);

        AX_STATE_UK_HOMING:
            TON_Exception.PT := T#0ms;
            TON_Exception.IN := NOT(MC_ReadStatus_0.Homing);

        (* States where the PLCopen state must be Standstill *)
        AX_STATE_STANDSTILL, AX_STATE_JOG_SS_HALTED:
            TON_Exception.PT := TIMEOUT_STATE_EXCEPTION;
            TON_Exception.IN := NOT(MC_ReadStatus_0.StandStill);

        AX_STATE_UK_STANDSTILL:
            TON_Exception.PT := T#0ms;
            TON_Exception.IN := NOT(MC_ReadStatus_0.StandStill);

        (* States where the PLCopen state must be ContinuousMotion *)
        AX_STATE_JOGGING_POS, AX_STATE_JOGGING_NEG,
        AX_STATE_MOVING_VELOCITY_0, AX_STATE_MOVING_VELOCITY_1:
            TON_Exception.PT := TIMEOUT_STATE_EXCEPTION;
            TON_Exception.IN := NOT(MC_ReadStatus_0.ContinuousMotion);

        AX_STATE_UK_CONTINUOUS_MOTION:
            TON_Exception.PT := T#0ms;
            TON_Exception.IN := NOT(MC_ReadStatus_0.ContinuousMotion);

        (* States where the PLCopen state must be DiscreteMotion *)
        AX_STATE_JOGGING_SS_POS, AX_STATE_JOGGING_SS_NEG, AX_STATE_HALTING_JOG,
        AX_STATE_MOVING_ABSOLUTE_0, AX_STATE_MOVING_ABSOLUTE_1,
        AX_STATE_MOVING_ADDITIVE_0, AX_STATE_MOVING_ADDITIVE_1,
        AX_STATE_HALTING_0, AX_STATE_HALTING_1:
            TON_Exception.PT := TIMEOUT_STATE_EXCEPTION;
            TON_Exception.IN := NOT(MC_ReadStatus_0.DiscreteMotion);

        AX_STATE_UK_DISCRETE_MOTION:
            TON_Exception.PT := T#0ms;
            TON_Exception.IN := NOT(MC_ReadStatus_0.DiscreteMotion);

        (* States where the PLCopen state must be SynchronizedMotion *)
		AX_STATE_MOVING_GEAR_0, AX_STATE_MOVING_GEAR_1:
			TON_Exception.PT := TIMEOUT_STATE_EXCEPTION;
			TON_Exception.IN := NOT(MC_ReadStatus_0.SynchronizedMotion);

		AX_STATE_UK_SYNCHRONIZED_MOTION:
            TON_Exception.PT := T#0ms;
            TON_Exception.IN := NOT(MC_ReadStatus_0.SynchronizedMotion);

        (* States where the PLCopen state must be Stopping *)
        AX_STATE_STOPPING:
            TON_Exception.PT := TIMEOUT_STATE_EXCEPTION;
            TON_Exception.IN := NOT(MC_ReadStatus_0.Stopping);

        AX_STATE_UK_STOPPING:
            TON_Exception.PT := T#0ms;
            TON_Exception.IN := NOT(MC_ReadStatus_0.Stopping);

        (* States where the PLCopen state must be ErrorStop *)
        AX_STATE_UK_ERROR_STOP:
            TON_Exception.PT := T#0ms;
            TON_Exception.IN := NOT(MC_ReadStatus_0.Errorstop);

        (* States which should be a fast transition *)
        AX_STATE_SWITCHING_OFF, AX_STATE_SWITCHING_ON:
            TON_Exception.PT := TIMEOUT_SWITCH_ON_OFF;
            TON_Exception.IN := TRUE;

        (* State where the PLCopen state must be determined immediately *)
        AX_STATE_UNKNOWN:
            TON_Exception.PT := T#0ms;
            TON_Exception.IN := TRUE;

        (* States where no state discrepancy is checked. No need to specify them *)
        ELSE

            (* ATTENTION! Program can stop working in these states *)
            (* To "protect" the program against hangs, add all newly *)
            (* created states wherever they should be in this CASE *)
            TON_Exception.IN := FALSE;

            (* In order not to get an error message, the following section can be commented out *)
            ErrorID := 50002;
            ClearErrorTexts;
            ErrorText[0] := 'At least an state has not been defined in the state supervisor';
            ErrorText[1] := 'ATTENTION: If a state is not defined, program may hang';
            AxisErrorState := AX_ERR_STATE_APP_ERROR;
            (* If desired, the following section can be uncommented to stop the axis as well *)
            //QuickStop;
            //AxisState := AX_STATE_UNKNOWN;

    END_CASE

    TON_Exception();

    (* Exception occurred *)
    IF TON_Exception.Q THEN
        TON_Exception.IN := FALSE;
        TON_Exception(); (* To be able to start right on the next cycle *)
        (* If the power should be off and MC_Power.Enable = 0   *)
        (* but the power is on because the Test Window did it,  *)
        (* since the MC_Power.Enable needs a negative edge to   *)
        (* switch it off, it must be enabled first              *)
        IF AxisState = AX_STATE_DISABLED THEN
            PowerOn;
        END_IF
        ResetExecutes;
        ResetMotionCommands;
        ResetJogCommands;
        DetermineState;
    END_IF

END_ACTION

(* Determines which is the actual PLCopen state *)
ACTION DetermineState:

    IF MC_ReadStatus_0.Valid THEN
        IF MC_ReadStatus_0.Disabled THEN
            (* If the power should be on and MC_Power.Enable = 1    *)
            (* but the power is off because the Test Window did it, *)
            (* since the MC_Power.Enable needs a positive edge to   *)
            (* switch it on, it must be disabled first              *)
            PowerOff;
            AxisState := AX_STATE_UK_DISABLED;
        ELSIF MC_ReadStatus_0.StandStill THEN
            AxisState := AX_STATE_UK_STANDSTILL;
        ELSIF MC_ReadStatus_0.Homing THEN
            AxisState := AX_STATE_UK_HOMING;
        ELSIF MC_ReadStatus_0.DiscreteMotion THEN
            AxisState := AX_STATE_UK_DISCRETE_MOTION;
        ELSIF MC_ReadStatus_0.ContinuousMotion THEN
            AxisState := AX_STATE_UK_CONTINUOUS_MOTION;
        ELSIF MC_ReadStatus_0.SynchronizedMotion THEN
            AxisState := AX_STATE_UK_SYNCHRONIZED_MOTION;
        ELSIF MC_ReadStatus_0.Stopping THEN
            AxisState := AX_STATE_UK_STOPPING;
        ELSIF MC_ReadStatus_0.Errorstop THEN
            AxisState := AX_STATE_UK_ERROR_STOP;
        ELSE
            AxisState := AX_STATE_UNKNOWN;
        END_IF
    ELSE
        AxisState := AX_STATE_UNKNOWN;
    END_IF

END_ACTION
```

### Library Logical/ExtPack/_Motion/AxisCtrl/AxisCtrl_v2/AxisFunc (IEC)

#### AxisFunc.fun - Exported functions and function blocks
```iecst
FUNCTION LoadDefaultStepperConfig : BOOL
	VAR_INPUT
		axisStepper : REFERENCE TO AxisCtrl_typ;
	END_VAR
END_FUNCTION

FUNCTION LoadDefaultServoConfig : BOOL
	VAR_INPUT
		axisServo : REFERENCE TO AxisCtrl_typ;
	END_VAR
END_FUNCTION
```

#### Drives.st
```iecst
(* Load Default configuration for Servodrives *)
FUNCTION LoadDefaultServoConfig

	axisServo.Parameter.Coms.ReadRatedTorque := TRUE;
	axisServo.Parameter.Coms.ReadMaxTorque := TRUE;

	LoadDefaultServoConfig := TRUE;

END_FUNCTION

(* Load Default configuration for Steppers *)
FUNCTION LoadDefaultStepperConfig

	axisStepper.Parameter.Init.xSendTorqueParams:=FALSE;
	axisStepper.Parameter.Coms.DisableReadingCurrent:=TRUE;
	axisStepper.Parameter.Coms.DisableReadingLagError:=TRUE;
	axisStepper.Parameter.Coms.DisableReadingTorque:=TRUE;
	axisStepper.Parameter.Coms.DisableReadingTemp:=TRUE;
	axisStepper.Parameter.Coms.ReadRatedTorque := FALSE;
	axisStepper.Parameter.Coms.ReadMaxTorque := FALSE;

	LoadDefaultStepperConfig := TRUE;

END_FUNCTION
```

### Program Logical/ExtPack/_Motion/AxisCtrl/AxisCtrl_v2/InitAxisControl

#### InitAxisControl.st
```iecst
PROGRAM _CYCLIC
	gIndexAxisCtrl	:= 1;
END_PROGRAM
```

### Inverter.typ
```iecst
TYPE
	AxisP66_Commands_typ : 	STRUCT  (*Control structure for ACOPOSinverter*)
		MovePositive : BOOL; (*Starts a movement in the positive direction*)
		MoveNegative : BOOL; (*Starts a movement in the negative direction*)
		Stop : BOOL; (*Stops the movement*)
		Reset : BOOL; (*Acknowledges and quits all errors*)
	END_STRUCT;
	AxisP66_Orders_typ : 	STRUCT  (*Control structure for ACOPOSinverter*)
		PowerOn : BOOL; (*Switches the power on*)
	END_STRUCT;
	AxisP66_ParametersHardware_typ : 	STRUCT
		CpuFamily : USINT;
		PowerLinkInterface : STRING[39]; (*Physical address of the Powerlink IF. For instance, 'SL1.IF3'*)
		Node : USINT; (*Inverter's Powerlink node*)
	END_STRUCT;
	AxisP66_Parameters_typ : 	STRUCT
		CommsType : CommsNetworkType_enum;
		Hardware : AxisP66_ParametersHardware_typ;
		Velocity : UINT := 200; (*[rpm]. Value of 200 by default in B&R code*)
		AccelerationTime : REAL := 3; (*[s]. Value of 3 by default in B&R code*)
		Type : InvType_enum;
		ControlMode : UINT := 0; (*Chose control mode: 1-Escalar, 0-Vectorial*)
		DecelerationTime : REAL := 3; (*[s]. Value of 3 by default in B&R code*)
	END_STRUCT;
	AxisP66_StatusHw_typ : 	STRUCT
		SerialNumber : UDINT;
		ModuleID : UDINT;
		HwVariant : UDINT;
		FwVersion : UDINT;
		ACPiSerialNumber : UDINT;
		ACPiModuleID : UDINT;
	END_STRUCT;
	AxisP66_Status_typ : 	STRUCT
		xAtSpeed : BOOL;
		ActVelocity : INT; (*[rpm]*)
		ActCurrent : REAL; (*[A]*)
		ActTorque : REAL; (*[Nm]*)
		ErrorID : UINT; (*Error number*)
		ErrorText : STRING[19]; (*Error description*)
		ErrorComms : BOOL; (*The comunication with the inverter is not working*)
		StatusDisabled : BOOL; (*The inverter is switched off*)
		StatusReady : BOOL; (*The inverter is ready to perform a movement*)
		StatusOperation : BOOL; (*The motor is powered*)
		StatusErrorStop : BOOL; (*The inverter has some error*)
		ReadyForOrders : BOOL; (*Powered OR Enabled*)
	END_STRUCT;
	AxisP66_ElecSignals_Out_typ : 	STRUCT
		xSpare : BOOL;
	END_STRUCT;
	AxisP66_ElecSignals_In_typ : 	STRUCT
		xBreakerOK : BOOL; (*EFI Signal: Circuit breaker protection OK*)
	END_STRUCT;
	AxisP66_ElecSignals_typ : 	STRUCT
		In : AxisP66_ElecSignals_In_typ;
		Out : AxisP66_ElecSignals_Out_typ;
	END_STRUCT;
	AxisP66_Signals_In_typ : 	STRUCT
		Hw : AxisP66_StatusHw_typ;
		Inputs : USINT;
		ModuleOk : BOOL; (*ModuleOk **)
		StatusWord : UINT; (*ETAD_Input **)
		ActualSpeed : INT; (*RFRD_Input [rpm] (encoderless estimation)*)
		ActualCurrent : UINT; (*LCR_Input (0.1A)*)
		ActualCurrentABB : INT; (*LCR_Input (0.001A)*)
		ActualTorque : INT; (*OTRN_Input (0.1Nm)*)
		ErrorID : UINT; (*LFT_Input*)
		DigitalInputs : UINT; (*Digital inputs in CanOpen. Reading an integer*)
		DigitalInput : ARRAY[0..7]OF BOOL; (*Digital inputs in Powerlink. Reading individually*)
		AnalogInput : ARRAY[0..2]OF INT;
		xBreakerOK : BOOL; (*EFI Signal: Circuit breaker protection OK*)
	END_STRUCT;
	AxisP66_Signals_Out_typ : 	STRUCT
		ControlWord : UINT; (*CMDD_Output **)
		DigitalOutputs : UINT; (*Digital inputs in CanOpen. Writing an integer*)
		DigitalOutput : ARRAY[0..2]OF BOOL; (*Digital inputs in Powerlink. Writing individually*)
		AnalogOutput : UINT;
		AnalogOutputSigned : INT; (*In CanOpen, Analog Output is INT not UINT*)
		SetSpeed : INT; (*LFRD_Output **)
		Acceleration : UINT; (*Just for CanOpen. In Powerlink sent by FunctionBlock*)
		Deceleration : UINT; (*Just for CanOpen. In Powerlink sent by FunctionBlock*)
		SetFrequency : INT;
		ControlMode : UINT; (*ControlMode_Output*)
		SpeedUnit : UINT; (*Velocity unit depending on the control mode.*)
		AccTimeVector : DINT;
		DecTimeVector : DINT;
		AccTimeScalar : DINT;
		DecTimeScalar : DINT;
		Reset : UINT;
	END_STRUCT;
	AxisP66_Signals_typ : 	STRUCT  (* * -> Compulsory*)
		In : AxisP66_Signals_In_typ;
		Out : AxisP66_Signals_Out_typ;
	END_STRUCT;
	AxisP66_typ : 	STRUCT  (*Control structure for ACOPOSinverter P66 & P67*)
		Commands : AxisP66_Commands_typ;
		Orders : AxisP66_Orders_typ;
		Parameters : AxisP66_Parameters_typ;
		Status : AxisP66_Status_typ;
		ElecSignals : AxisP66_ElecSignals_typ;
		DigitalInput : ARRAY[0..7]OF BOOL;
		DigitalOutput : ARRAY[0..2]OF BOOL;
		AnalogInput : ARRAY[0..2]OF INT;
		AnalogOutput : UINT;
	END_STRUCT;
END_TYPE
```

### Program Logical/ExtPack/_Motion/InverterCtrl/InverterCtrl_v1/InverterCtrl

#### ErrorTable.st
```iecst
(********************************************************************
 * COPYRIGHT -- Bernecker + Rainer
 ********************************************************************
 * Program: I66Ctrl
 * File: ErrorTable.st
 * Author: tresensa
 * Created: May 09, 2014
 ********************************************************************
 * Implementation of program InvCtrl
 ********************************************************************)

(*Writes the error table*)
ACTION ErrorTable:

	ERROR_TEXT[0] := 'NOF';
	//ERROR_TEXT[1] := 'InF'; // Not in the table.
	ERROR_TEXT[2] := 'EEF1';
	ERROR_TEXT[3] := 'CFF';
	ERROR_TEXT[4] := 'CFI';
	ERROR_TEXT[5] := 'SLF1';
	ERROR_TEXT[6] := 'ILF';
	ERROR_TEXT[7] := 'CnF';
	ERROR_TEXT[8] := 'EPF1';
	ERROR_TEXT[9] := 'OCF';
	ERROR_TEXT[10] := 'CrF';
	ERROR_TEXT[11] := 'SRF'; // Originally: SRF.

	ERROR_TEXT[16] := 'OHF';
	ERROR_TEXT[17] := 'OLF';
	ERROR_TEXT[18] := 'ObF';
	ERROR_TEXT[19] := 'OSF';
	ERROR_TEXT[20] := 'OPF1';
	ERROR_TEXT[21] := 'PHF';
	ERROR_TEXT[22] := 'USF';
	ERROR_TEXT[23] := 'SCF1';
	ERROR_TEXT[24] := 'SOF';
	ERROR_TEXT[25] := 'tnF';
	ERROR_TEXT[26] := 'InF1';
	ERROR_TEXT[27] := 'InF2';
	ERROR_TEXT[28] := 'InF3';
	ERROR_TEXT[29] := 'InF4';
	ERROR_TEXT[30] := 'EEF2';
	//ERROR_TEXT[31] := 'SCF2'; // Not in the table.
	ERROR_TEXT[32] := 'SCF3';
	ERROR_TEXT[33] := 'OPF2';
	ERROR_TEXT[34] := 'COF';
	ERROR_TEXT[35] := 'bLF';

	ERROR_TEXT[38] := 'EPF2';

	ERROR_TEXT[41] := 'brF';
	ERROR_TEXT[42] := 'SLF2';
	//ERROR_TEXT[43] := 'ECF'; // Not in the table.
	ERROR_TEXT[44] := 'SSF';
	ERROR_TEXT[45] := 'SLF3';
	//ERROR_TEXT[46] := 'PrF'; // Not in the table.

	ERROR_TEXT[49] := 'PtFL';
	ERROR_TEXT[50] := 'OtFL';
	ERROR_TEXT[51] := 'InF9';
	ERROR_TEXT[52] := 'InFA';
	ERROR_TEXT[53] := 'InFb';
	ERROR_TEXT[54] := 'tJF';
	ERROR_TEXT[55] := 'SCF4';
	ERROR_TEXT[56] := 'SCF5';
	//ERROR_TEXT[57] := 'SrF'; // Not in the table.
	ERROR_TEXT[58] := 'FCF1';
	ERROR_TEXT[59] := 'FCF2';

	//ERROR_TEXT[61] := 'AI2F'; // Not in the table.

	ERROR_TEXT[64] := 'LCF';

	//ERROR_TEXT[66] := 'dCF'; // Not in the table.
	ERROR_TEXT[67] := 'HdF';
	ERROR_TEXT[68] := 'InF6';
	ERROR_TEXT[69] := 'InFE';

	ERROR_TEXT[71] := 'LFF3';

	ERROR_TEXT[73] := 'HCF';

	ERROR_TEXT[76] := 'dLF';
	ERROR_TEXT[77] := 'CFI2';

	ERROR_TEXT[99] := 'CSF';
	ERROR_TEXT[100] := 'ULF';
	ERROR_TEXT[101] := 'OLF'; // Originally: OLC.

	ERROR_TEXT[105] := 'ASF';

	ERROR_TEXT[107] := 'SAFF';
	//ERROR_TEXT[108] := 'FbE'; // Not in the table.
	//ERROR_TEXT[109] := 'FbES'; // Not in the table.

END_ACTION
```
